REGION Network 2
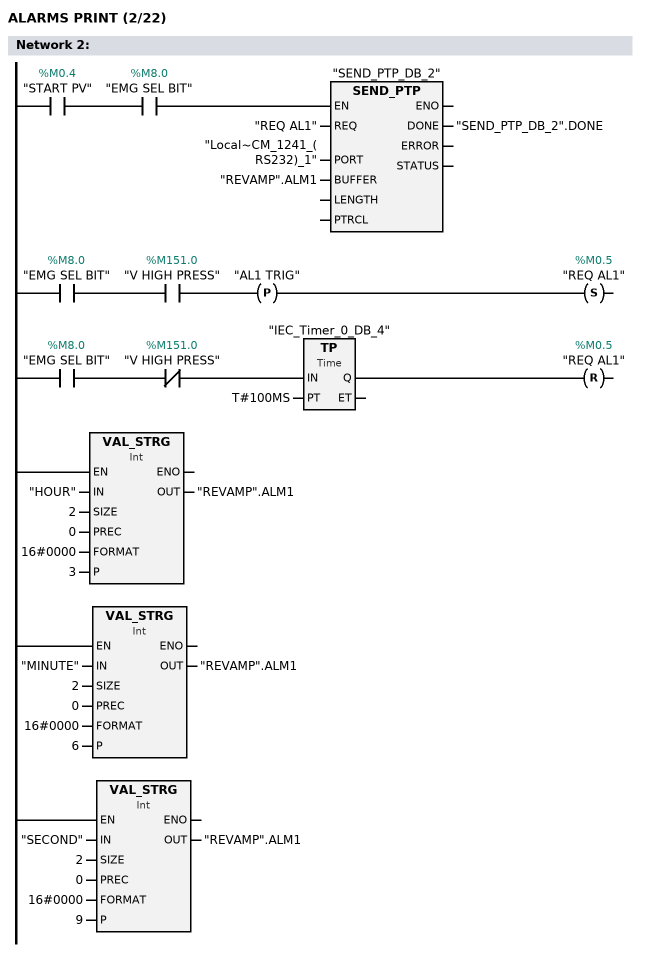
   RUNG wire#powerrail
      Contact( "START PV" )
      Contact( "EMG SEL BIT" )
      "SEND_PTP_DB_2".SEND_PTP(REQ := "REQ AL1", PORT := "Local~CM_1241_(RS232)_1", BUFFER := "REVAMP".ALM1, LENGTH :=, PTRCL :=, DONE => "SEND_PTP_DB_2".DONE, ERROR =>, STATUS =>)
   END_RUNG
   RUNG wire#powerrail
      Contact( "EMG SEL BIT" )
      Contact( "V HIGH PRESS" )
      P_Trig( "AL1 TRIG" )
      S_Coil( "REQ AL1" )
   END_RUNG
   RUNG wire#powerrail
      Contact( "EMG SEL BIT" )
      I_Contact( "V HIGH PRESS" )
      { S7_Templates := "time_type := Time" } "IEC_Timer_0_DB_4".TP(pt := T#100MS, et =>)
      R_Coil( "REQ AL1" )
   END_RUNG
   RUNG wire#powerrail
      { S7_Templates := "[value_type := Int, str_type := String]" } VAL_STRG(IN := "HOUR", SIZE := 2, PREC := 0, FORMAT := 16#0000, P := 3, OUT => "REVAMP".ALM1)
   END_RUNG
   RUNG wire#powerrail
      { S7_Templates := "[value_type := Int, str_type := String]" } VAL_STRG(IN := "MINUTE", SIZE := 2, PREC := 0, FORMAT := 16#0000, P := 6, OUT => "REVAMP".ALM1)
   END_RUNG
   RUNG wire#powerrail
      { S7_Templates := "[value_type := Int, str_type := String]" } VAL_STRG(IN := "SECOND", SIZE := 2, PREC := 0, FORMAT := 16#0000, P := 9, OUT => "REVAMP".ALM1)
   END_RUNG
   // the same network as SCL:
   IF "START PV" AND "EMG SEL BIT" THEN
       "SEND_PTP_DB_2"(REQ := "REQ AL1",   // SEND_PTP
                       PORT := "Local~CM_1241_(RS232)_1",
                       BUFFER := "REVAMP".ALM1,
                       DONE => "SEND_PTP_DB_2".DONE);
   END_IF;
   #_w1 := "EMG SEL BIT" AND "V HIGH PRESS";
   #_w2 := #_w1 AND NOT "AL1 TRIG";   // rising edge
   "AL1 TRIG" := #_w1;
   IF #_w2 THEN "REQ AL1" := TRUE; END_IF;
   "IEC_Timer_0_DB_4".TP(IN := "EMG SEL BIT" AND NOT "V HIGH PRESS", PT := T#100MS);
   IF "IEC_Timer_0_DB_4".Q THEN "REQ AL1" := FALSE; END_IF;
   VAL_STRG(IN := "HOUR", SIZE := 2, PREC := 0, FORMAT := 16#0000, P := 3, OUT => "REVAMP".ALM1);
   VAL_STRG(IN := "MINUTE", SIZE := 2, PREC := 0, FORMAT := 16#0000, P := 6, OUT => "REVAMP".ALM1);
   VAL_STRG(IN := "SECOND", SIZE := 2, PREC := 0, FORMAT := 16#0000, P := 9, OUT => "REVAMP".ALM1);
END_REGION

REGION Network 3
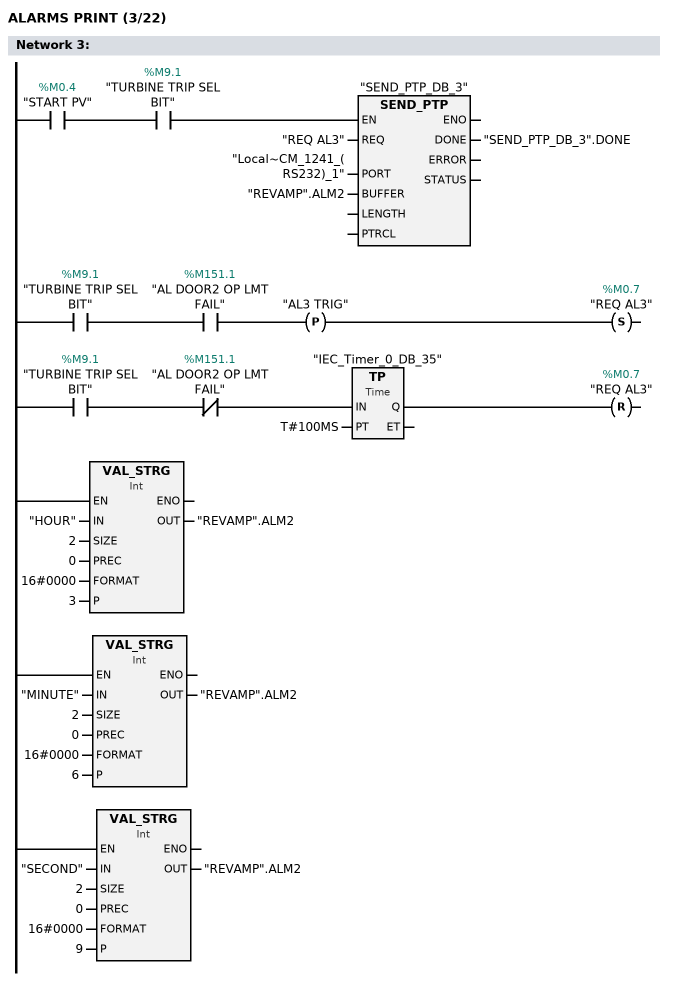
   RUNG wire#powerrail
      Contact( "START PV" )
      Contact( "TURBINE TRIP SEL BIT" )
      "SEND_PTP_DB_3".SEND_PTP(REQ := "REQ AL3", PORT := "Local~CM_1241_(RS232)_1", BUFFER := "REVAMP".ALM2, LENGTH :=, PTRCL :=, DONE => "SEND_PTP_DB_3".DONE, ERROR =>, STATUS =>)
   END_RUNG
   RUNG wire#powerrail
      Contact( "TURBINE TRIP SEL BIT" )
      Contact( "AL DOOR2 OP LMT FAIL" )
      P_Trig( "AL3 TRIG" )
      S_Coil( "REQ AL3" )
   END_RUNG
   RUNG wire#powerrail
      Contact( "TURBINE TRIP SEL BIT" )
      I_Contact( "AL DOOR2 OP LMT FAIL" )
      { S7_Templates := "time_type := Time" } "IEC_Timer_0_DB_35".TP(pt := T#100MS, et =>)
      R_Coil( "REQ AL3" )
   END_RUNG
   RUNG wire#powerrail
      { S7_Templates := "[value_type := Int, str_type := String]" } VAL_STRG(IN := "HOUR", SIZE := 2, PREC := 0, FORMAT := 16#0000, P := 3, OUT => "REVAMP".ALM2)
   END_RUNG
   RUNG wire#powerrail
      { S7_Templates := "[value_type := Int, str_type := String]" } VAL_STRG(IN := "MINUTE", SIZE := 2, PREC := 0, FORMAT := 16#0000, P := 6, OUT => "REVAMP".ALM2)
   END_RUNG
   RUNG wire#powerrail
      { S7_Templates := "[value_type := Int, str_type := String]" } VAL_STRG(IN := "SECOND", SIZE := 2, PREC := 0, FORMAT := 16#0000, P := 9, OUT => "REVAMP".ALM2)
   END_RUNG
   // the same network as SCL:
   IF "START PV" AND "TURBINE TRIP SEL BIT" THEN
       "SEND_PTP_DB_3"(REQ := "REQ AL3",   // SEND_PTP
                       PORT := "Local~CM_1241_(RS232)_1",
                       BUFFER := "REVAMP".ALM2,
                       DONE => "SEND_PTP_DB_3".DONE);
   END_IF;
   #_w1 := "TURBINE TRIP SEL BIT" AND "AL DOOR2 OP LMT FAIL";
   #_w2 := #_w1 AND NOT "AL3 TRIG";   // rising edge
   "AL3 TRIG" := #_w1;
   IF #_w2 THEN "REQ AL3" := TRUE; END_IF;
   "IEC_Timer_0_DB_35".TP(IN := "TURBINE TRIP SEL BIT" AND NOT "AL DOOR2 OP LMT FAIL", PT := T#100MS);
   IF "IEC_Timer_0_DB_35".Q THEN "REQ AL3" := FALSE; END_IF;
   VAL_STRG(IN := "HOUR", SIZE := 2, PREC := 0, FORMAT := 16#0000, P := 3, OUT => "REVAMP".ALM2);
   VAL_STRG(IN := "MINUTE", SIZE := 2, PREC := 0, FORMAT := 16#0000, P := 6, OUT => "REVAMP".ALM2);
   VAL_STRG(IN := "SECOND", SIZE := 2, PREC := 0, FORMAT := 16#0000, P := 9, OUT => "REVAMP".ALM2);
END_REGION

REGION Network 4
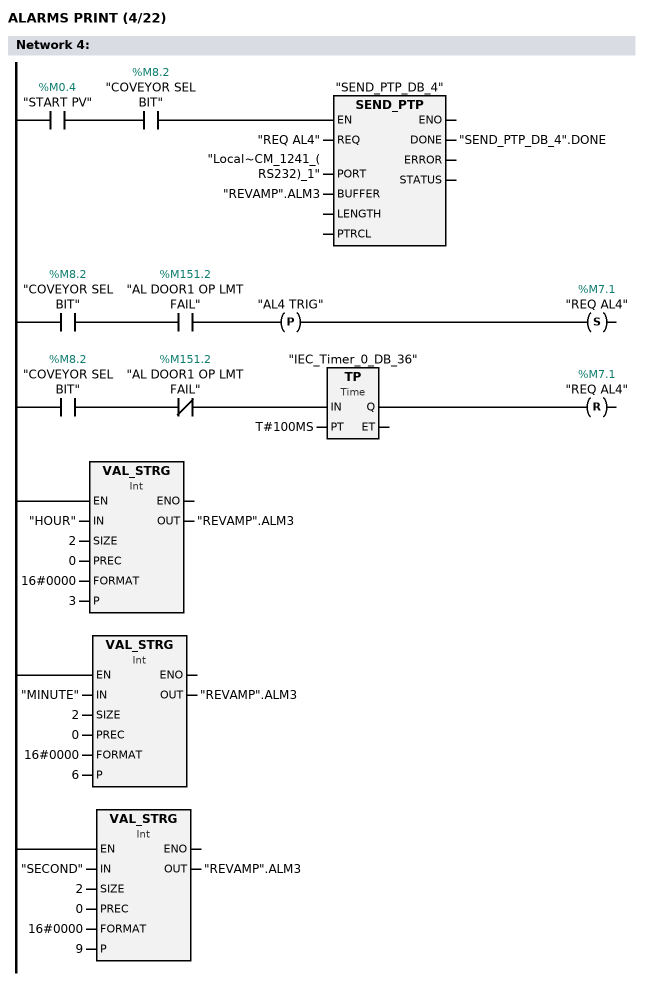
   RUNG wire#powerrail
      Contact( "START PV" )
      Contact( "COVEYOR SEL BIT" )
      "SEND_PTP_DB_4".SEND_PTP(REQ := "REQ AL4", PORT := "Local~CM_1241_(RS232)_1", BUFFER := "REVAMP".ALM3, LENGTH :=, PTRCL :=, DONE => "SEND_PTP_DB_4".DONE, ERROR =>, STATUS =>)
   END_RUNG
   RUNG wire#powerrail
      Contact( "COVEYOR SEL BIT" )
      Contact( "AL DOOR1 OP LMT FAIL" )
      P_Trig( "AL4 TRIG" )
      S_Coil( "REQ AL4" )
   END_RUNG
   RUNG wire#powerrail
      Contact( "COVEYOR SEL BIT" )
      I_Contact( "AL DOOR1 OP LMT FAIL" )
      { S7_Templates := "time_type := Time" } "IEC_Timer_0_DB_36".TP(pt := T#100MS, et =>)
      R_Coil( "REQ AL4" )
   END_RUNG
   RUNG wire#powerrail
      { S7_Templates := "[value_type := Int, str_type := String]" } VAL_STRG(IN := "HOUR", SIZE := 2, PREC := 0, FORMAT := 16#0000, P := 3, OUT => "REVAMP".ALM3)
   END_RUNG
   RUNG wire#powerrail
      { S7_Templates := "[value_type := Int, str_type := String]" } VAL_STRG(IN := "MINUTE", SIZE := 2, PREC := 0, FORMAT := 16#0000, P := 6, OUT => "REVAMP".ALM3)
   END_RUNG
   RUNG wire#powerrail
      { S7_Templates := "[value_type := Int, str_type := String]" } VAL_STRG(IN := "SECOND", SIZE := 2, PREC := 0, FORMAT := 16#0000, P := 9, OUT => "REVAMP".ALM3)
   END_RUNG
   // the same network as SCL:
   IF "START PV" AND "COVEYOR SEL BIT" THEN
       "SEND_PTP_DB_4"(REQ := "REQ AL4",   // SEND_PTP
                       PORT := "Local~CM_1241_(RS232)_1",
                       BUFFER := "REVAMP".ALM3,
                       DONE => "SEND_PTP_DB_4".DONE);
   END_IF;
   #_w1 := "COVEYOR SEL BIT" AND "AL DOOR1 OP LMT FAIL";
   #_w2 := #_w1 AND NOT "AL4 TRIG";   // rising edge
   "AL4 TRIG" := #_w1;
   IF #_w2 THEN "REQ AL4" := TRUE; END_IF;
   "IEC_Timer_0_DB_36".TP(IN := "COVEYOR SEL BIT" AND NOT "AL DOOR1 OP LMT FAIL", PT := T#100MS);
   IF "IEC_Timer_0_DB_36".Q THEN "REQ AL4" := FALSE; END_IF;
   VAL_STRG(IN := "HOUR", SIZE := 2, PREC := 0, FORMAT := 16#0000, P := 3, OUT => "REVAMP".ALM3);
   VAL_STRG(IN := "MINUTE", SIZE := 2, PREC := 0, FORMAT := 16#0000, P := 6, OUT => "REVAMP".ALM3);
   VAL_STRG(IN := "SECOND", SIZE := 2, PREC := 0, FORMAT := 16#0000, P := 9, OUT => "REVAMP".ALM3);
END_REGION

REGION Network 5
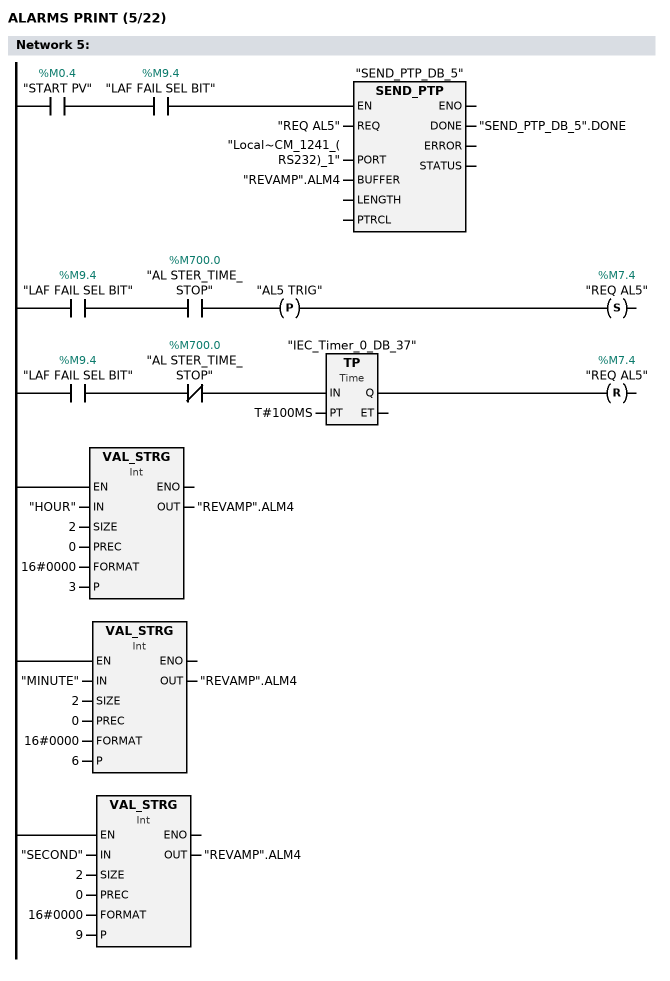
   RUNG wire#powerrail
      Contact( "START PV" )
      Contact( "LAF FAIL SEL BIT" )
      "SEND_PTP_DB_5".SEND_PTP(REQ := "REQ AL5", PORT := "Local~CM_1241_(RS232)_1", BUFFER := "REVAMP".ALM4, LENGTH :=, PTRCL :=, DONE => "SEND_PTP_DB_5".DONE, ERROR =>, STATUS =>)
   END_RUNG
   RUNG wire#powerrail
      Contact( "LAF FAIL SEL BIT" )
      Contact( "AL STER_TIME_STOP" )
      P_Trig( "AL5 TRIG" )
      S_Coil( "REQ AL5" )
   END_RUNG
   RUNG wire#powerrail
      Contact( "LAF FAIL SEL BIT" )
      I_Contact( "AL STER_TIME_STOP" )
      { S7_Templates := "time_type := Time" } "IEC_Timer_0_DB_37".TP(pt := T#100MS, et =>)
      R_Coil( "REQ AL5" )
   END_RUNG
   RUNG wire#powerrail
      { S7_Templates := "[value_type := Int, str_type := String]" } VAL_STRG(IN := "HOUR", SIZE := 2, PREC := 0, FORMAT := 16#0000, P := 3, OUT => "REVAMP".ALM4)
   END_RUNG
   RUNG wire#powerrail
      { S7_Templates := "[value_type := Int, str_type := String]" } VAL_STRG(IN := "MINUTE", SIZE := 2, PREC := 0, FORMAT := 16#0000, P := 6, OUT => "REVAMP".ALM4)
   END_RUNG
   RUNG wire#powerrail
      { S7_Templates := "[value_type := Int, str_type := String]" } VAL_STRG(IN := "SECOND", SIZE := 2, PREC := 0, FORMAT := 16#0000, P := 9, OUT => "REVAMP".ALM4)
   END_RUNG
   // the same network as SCL:
   IF "START PV" AND "LAF FAIL SEL BIT" THEN
       "SEND_PTP_DB_5"(REQ := "REQ AL5",   // SEND_PTP
                       PORT := "Local~CM_1241_(RS232)_1",
                       BUFFER := "REVAMP".ALM4,
                       DONE => "SEND_PTP_DB_5".DONE);
   END_IF;
   #_w1 := "LAF FAIL SEL BIT" AND "AL STER_TIME_STOP";
   #_w2 := #_w1 AND NOT "AL5 TRIG";   // rising edge
   "AL5 TRIG" := #_w1;
   IF #_w2 THEN "REQ AL5" := TRUE; END_IF;
   "IEC_Timer_0_DB_37".TP(IN := "LAF FAIL SEL BIT" AND NOT "AL STER_TIME_STOP", PT := T#100MS);
   IF "IEC_Timer_0_DB_37".Q THEN "REQ AL5" := FALSE; END_IF;
   VAL_STRG(IN := "HOUR", SIZE := 2, PREC := 0, FORMAT := 16#0000, P := 3, OUT => "REVAMP".ALM4);
   VAL_STRG(IN := "MINUTE", SIZE := 2, PREC := 0, FORMAT := 16#0000, P := 6, OUT => "REVAMP".ALM4);
   VAL_STRG(IN := "SECOND", SIZE := 2, PREC := 0, FORMAT := 16#0000, P := 9, OUT => "REVAMP".ALM4);
END_REGION

REGION Network 6
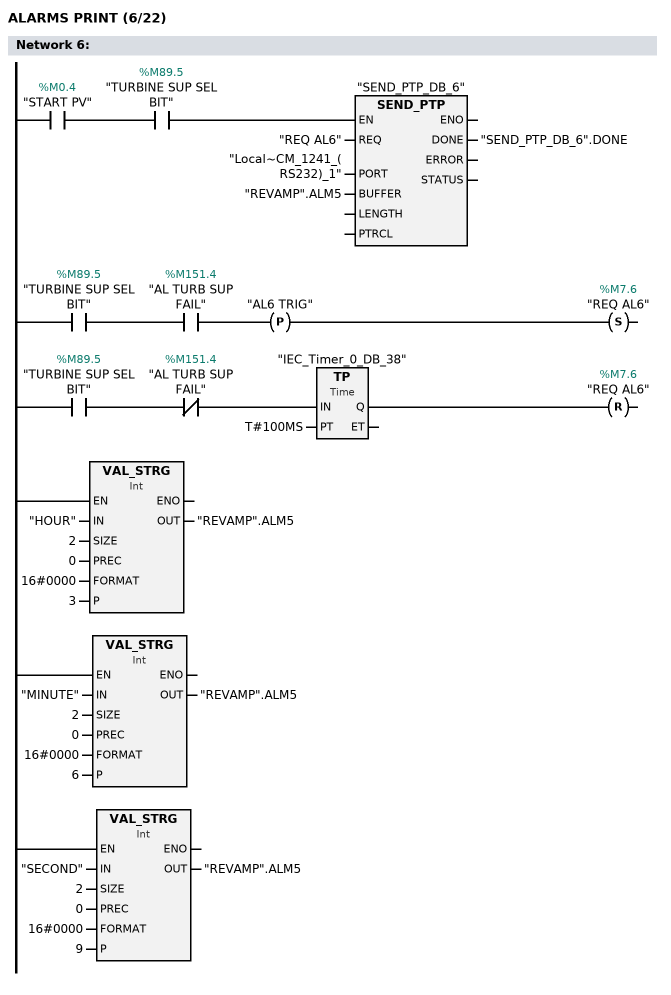
   RUNG wire#powerrail
      Contact( "START PV" )
      Contact( "TURBINE SUP SEL BIT" )
      "SEND_PTP_DB_6".SEND_PTP(REQ := "REQ AL6", PORT := "Local~CM_1241_(RS232)_1", BUFFER := "REVAMP".ALM5, LENGTH :=, PTRCL :=, DONE => "SEND_PTP_DB_6".DONE, ERROR =>, STATUS =>)
   END_RUNG
   RUNG wire#powerrail
      Contact( "TURBINE SUP SEL BIT" )
      Contact( "AL TURB SUP FAIL" )
      P_Trig( "AL6 TRIG" )
      S_Coil( "REQ AL6" )
   END_RUNG
   RUNG wire#powerrail
      Contact( "TURBINE SUP SEL BIT" )
      I_Contact( "AL TURB SUP FAIL" )
      { S7_Templates := "time_type := Time" } "IEC_Timer_0_DB_38".TP(pt := T#100MS, et =>)
      R_Coil( "REQ AL6" )
   END_RUNG
   RUNG wire#powerrail
      { S7_Templates := "[value_type := Int, str_type := String]" } VAL_STRG(IN := "HOUR", SIZE := 2, PREC := 0, FORMAT := 16#0000, P := 3, OUT => "REVAMP".ALM5)
   END_RUNG
   RUNG wire#powerrail
      { S7_Templates := "[value_type := Int, str_type := String]" } VAL_STRG(IN := "MINUTE", SIZE := 2, PREC := 0, FORMAT := 16#0000, P := 6, OUT => "REVAMP".ALM5)
   END_RUNG
   RUNG wire#powerrail
      { S7_Templates := "[value_type := Int, str_type := String]" } VAL_STRG(IN := "SECOND", SIZE := 2, PREC := 0, FORMAT := 16#0000, P := 9, OUT => "REVAMP".ALM5)
   END_RUNG
   // the same network as SCL:
   IF "START PV" AND "TURBINE SUP SEL BIT" THEN
       "SEND_PTP_DB_6"(REQ := "REQ AL6",   // SEND_PTP
                       PORT := "Local~CM_1241_(RS232)_1",
                       BUFFER := "REVAMP".ALM5,
                       DONE => "SEND_PTP_DB_6".DONE);
   END_IF;
   #_w1 := "TURBINE SUP SEL BIT" AND "AL TURB SUP FAIL";
   #_w2 := #_w1 AND NOT "AL6 TRIG";   // rising edge
   "AL6 TRIG" := #_w1;
   IF #_w2 THEN "REQ AL6" := TRUE; END_IF;
   "IEC_Timer_0_DB_38".TP(IN := "TURBINE SUP SEL BIT" AND NOT "AL TURB SUP FAIL", PT := T#100MS);
   IF "IEC_Timer_0_DB_38".Q THEN "REQ AL6" := FALSE; END_IF;
   VAL_STRG(IN := "HOUR", SIZE := 2, PREC := 0, FORMAT := 16#0000, P := 3, OUT => "REVAMP".ALM5);
   VAL_STRG(IN := "MINUTE", SIZE := 2, PREC := 0, FORMAT := 16#0000, P := 6, OUT => "REVAMP".ALM5);
   VAL_STRG(IN := "SECOND", SIZE := 2, PREC := 0, FORMAT := 16#0000, P := 9, OUT => "REVAMP".ALM5);
END_REGION

REGION Network 7
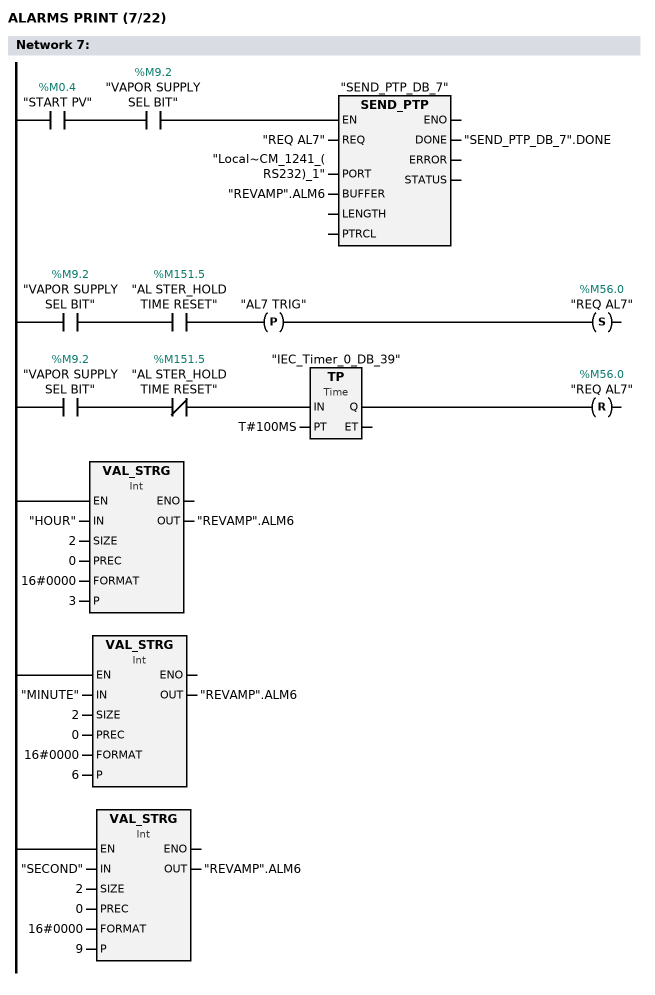
   RUNG wire#powerrail
      Contact( "START PV" )
      Contact( "VAPOR SUPPLY SEL BIT" )
      "SEND_PTP_DB_7".SEND_PTP(REQ := "REQ AL7", PORT := "Local~CM_1241_(RS232)_1", BUFFER := "REVAMP".ALM6, LENGTH :=, PTRCL :=, DONE => "SEND_PTP_DB_7".DONE, ERROR =>, STATUS =>)
   END_RUNG
   RUNG wire#powerrail
      Contact( "VAPOR SUPPLY SEL BIT" )
      Contact( "AL STER_HOLD TIME RESET" )
      P_Trig( "AL7 TRIG" )
      S_Coil( "REQ AL7" )
   END_RUNG
   RUNG wire#powerrail
      Contact( "VAPOR SUPPLY SEL BIT" )
      I_Contact( "AL STER_HOLD TIME RESET" )
      { S7_Templates := "time_type := Time" } "IEC_Timer_0_DB_39".TP(pt := T#100MS, et =>)
      R_Coil( "REQ AL7" )
   END_RUNG
   RUNG wire#powerrail
      { S7_Templates := "[value_type := Int, str_type := String]" } VAL_STRG(IN := "HOUR", SIZE := 2, PREC := 0, FORMAT := 16#0000, P := 3, OUT => "REVAMP".ALM6)
   END_RUNG
   RUNG wire#powerrail
      { S7_Templates := "[value_type := Int, str_type := String]" } VAL_STRG(IN := "MINUTE", SIZE := 2, PREC := 0, FORMAT := 16#0000, P := 6, OUT => "REVAMP".ALM6)
   END_RUNG
   RUNG wire#powerrail
      { S7_Templates := "[value_type := Int, str_type := String]" } VAL_STRG(IN := "SECOND", SIZE := 2, PREC := 0, FORMAT := 16#0000, P := 9, OUT => "REVAMP".ALM6)
   END_RUNG
   // the same network as SCL:
   IF "START PV" AND "VAPOR SUPPLY SEL BIT" THEN
       "SEND_PTP_DB_7"(REQ := "REQ AL7",   // SEND_PTP
                       PORT := "Local~CM_1241_(RS232)_1",
                       BUFFER := "REVAMP".ALM6,
                       DONE => "SEND_PTP_DB_7".DONE);
   END_IF;
   #_w1 := "VAPOR SUPPLY SEL BIT" AND "AL STER_HOLD TIME RESET";
   #_w2 := #_w1 AND NOT "AL7 TRIG";   // rising edge
   "AL7 TRIG" := #_w1;
   IF #_w2 THEN "REQ AL7" := TRUE; END_IF;
   "IEC_Timer_0_DB_39".TP(IN := "VAPOR SUPPLY SEL BIT" AND NOT "AL STER_HOLD TIME RESET", PT := T#100MS);
   IF "IEC_Timer_0_DB_39".Q THEN "REQ AL7" := FALSE; END_IF;
   VAL_STRG(IN := "HOUR", SIZE := 2, PREC := 0, FORMAT := 16#0000, P := 3, OUT => "REVAMP".ALM6);
   VAL_STRG(IN := "MINUTE", SIZE := 2, PREC := 0, FORMAT := 16#0000, P := 6, OUT => "REVAMP".ALM6);
   VAL_STRG(IN := "SECOND", SIZE := 2, PREC := 0, FORMAT := 16#0000, P := 9, OUT => "REVAMP".ALM6);
END_REGION

REGION Network 8
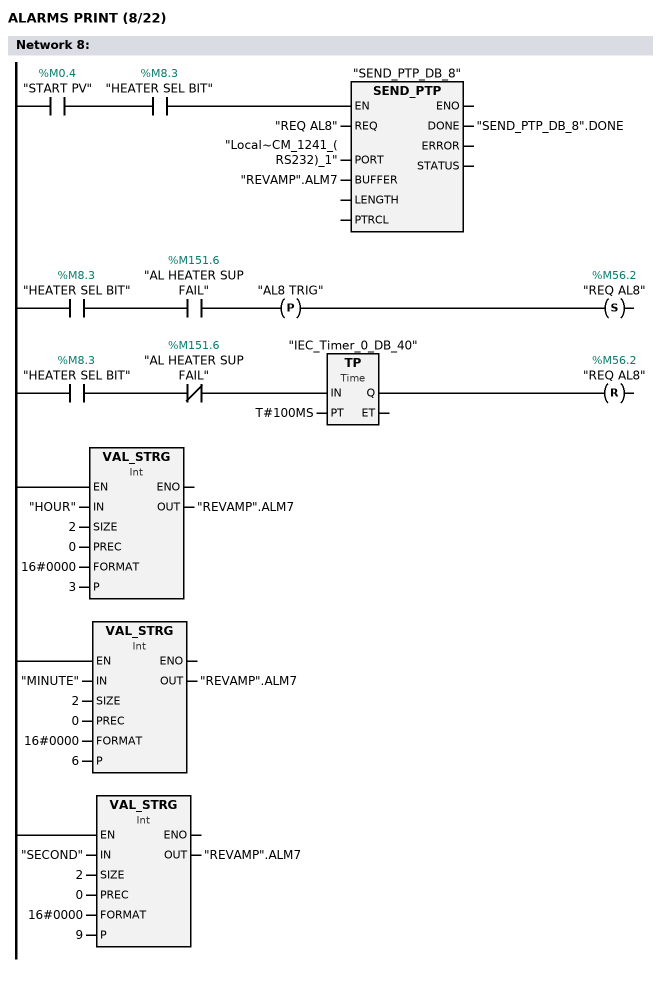
   RUNG wire#powerrail
      Contact( "START PV" )
      Contact( "HEATER SEL BIT" )
      "SEND_PTP_DB_8".SEND_PTP(REQ := "REQ AL8", PORT := "Local~CM_1241_(RS232)_1", BUFFER := "REVAMP".ALM7, LENGTH :=, PTRCL :=, DONE => "SEND_PTP_DB_8".DONE, ERROR =>, STATUS =>)
   END_RUNG
   RUNG wire#powerrail
      Contact( "HEATER SEL BIT" )
      Contact( "AL HEATER SUP FAIL" )
      P_Trig( "AL8 TRIG" )
      S_Coil( "REQ AL8" )
   END_RUNG
   RUNG wire#powerrail
      Contact( "HEATER SEL BIT" )
      I_Contact( "AL HEATER SUP FAIL" )
      { S7_Templates := "time_type := Time" } "IEC_Timer_0_DB_40".TP(pt := T#100MS, et =>)
      R_Coil( "REQ AL8" )
   END_RUNG
   RUNG wire#powerrail
      { S7_Templates := "[value_type := Int, str_type := String]" } VAL_STRG(IN := "HOUR", SIZE := 2, PREC := 0, FORMAT := 16#0000, P := 3, OUT => "REVAMP".ALM7)
   END_RUNG
   RUNG wire#powerrail
      { S7_Templates := "[value_type := Int, str_type := String]" } VAL_STRG(IN := "MINUTE", SIZE := 2, PREC := 0, FORMAT := 16#0000, P := 6, OUT => "REVAMP".ALM7)
   END_RUNG
   RUNG wire#powerrail
      { S7_Templates := "[value_type := Int, str_type := String]" } VAL_STRG(IN := "SECOND", SIZE := 2, PREC := 0, FORMAT := 16#0000, P := 9, OUT => "REVAMP".ALM7)
   END_RUNG
   // the same network as SCL:
   IF "START PV" AND "HEATER SEL BIT" THEN
       "SEND_PTP_DB_8"(REQ := "REQ AL8",   // SEND_PTP
                       PORT := "Local~CM_1241_(RS232)_1",
                       BUFFER := "REVAMP".ALM7,
                       DONE => "SEND_PTP_DB_8".DONE);
   END_IF;
   #_w1 := "HEATER SEL BIT" AND "AL HEATER SUP FAIL";
   #_w2 := #_w1 AND NOT "AL8 TRIG";   // rising edge
   "AL8 TRIG" := #_w1;
   IF #_w2 THEN "REQ AL8" := TRUE; END_IF;
   "IEC_Timer_0_DB_40".TP(IN := "HEATER SEL BIT" AND NOT "AL HEATER SUP FAIL", PT := T#100MS);
   IF "IEC_Timer_0_DB_40".Q THEN "REQ AL8" := FALSE; END_IF;
   VAL_STRG(IN := "HOUR", SIZE := 2, PREC := 0, FORMAT := 16#0000, P := 3, OUT => "REVAMP".ALM7);
   VAL_STRG(IN := "MINUTE", SIZE := 2, PREC := 0, FORMAT := 16#0000, P := 6, OUT => "REVAMP".ALM7);
   VAL_STRG(IN := "SECOND", SIZE := 2, PREC := 0, FORMAT := 16#0000, P := 9, OUT => "REVAMP".ALM7);
END_REGION

REGION Network 9
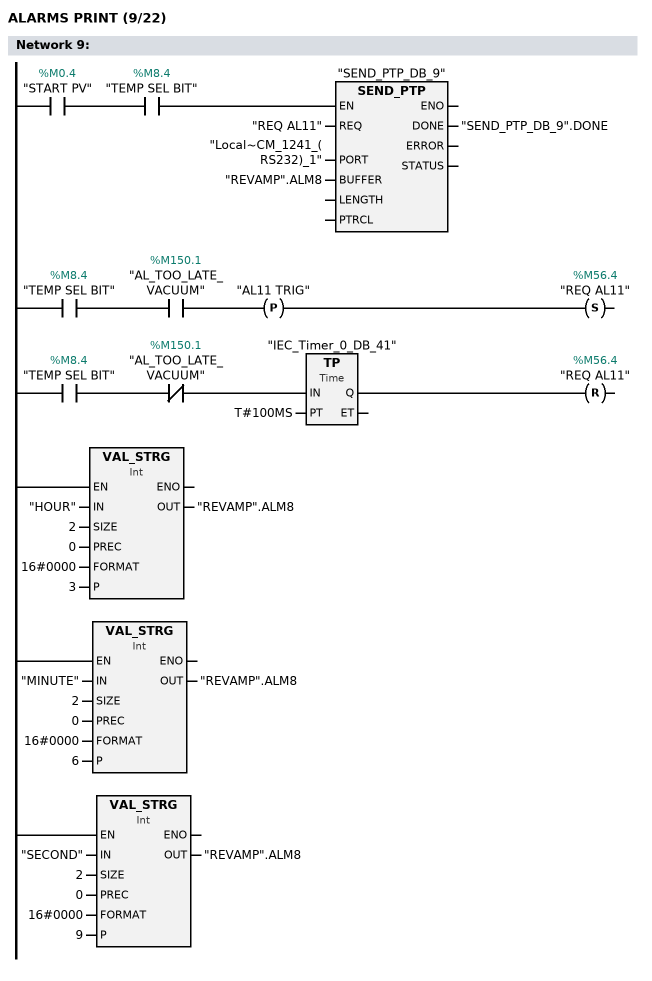
   RUNG wire#powerrail
      Contact( "START PV" )
      Contact( "TEMP SEL BIT" )
      "SEND_PTP_DB_9".SEND_PTP(REQ := "REQ AL11", PORT := "Local~CM_1241_(RS232)_1", BUFFER := "REVAMP".ALM8, LENGTH :=, PTRCL :=, DONE => "SEND_PTP_DB_9".DONE, ERROR =>, STATUS =>)
   END_RUNG
   RUNG wire#powerrail
      Contact( "TEMP SEL BIT" )
      Contact( "AL_TOO_LATE_VACUUM" )
      P_Trig( "AL11 TRIG" )
      S_Coil( "REQ AL11" )
   END_RUNG
   RUNG wire#powerrail
      Contact( "TEMP SEL BIT" )
      I_Contact( "AL_TOO_LATE_VACUUM" )
      { S7_Templates := "time_type := Time" } "IEC_Timer_0_DB_41".TP(pt := T#100MS, et =>)
      R_Coil( "REQ AL11" )
   END_RUNG
   RUNG wire#powerrail
      { S7_Templates := "[value_type := Int, str_type := String]" } VAL_STRG(IN := "HOUR", SIZE := 2, PREC := 0, FORMAT := 16#0000, P := 3, OUT => "REVAMP".ALM8)
   END_RUNG
   RUNG wire#powerrail
      { S7_Templates := "[value_type := Int, str_type := String]" } VAL_STRG(IN := "MINUTE", SIZE := 2, PREC := 0, FORMAT := 16#0000, P := 6, OUT => "REVAMP".ALM8)
   END_RUNG
   RUNG wire#powerrail
      { S7_Templates := "[value_type := Int, str_type := String]" } VAL_STRG(IN := "SECOND", SIZE := 2, PREC := 0, FORMAT := 16#0000, P := 9, OUT => "REVAMP".ALM8)
   END_RUNG
   // the same network as SCL:
   IF "START PV" AND "TEMP SEL BIT" THEN
       "SEND_PTP_DB_9"(REQ := "REQ AL11",   // SEND_PTP
                       PORT := "Local~CM_1241_(RS232)_1",
                       BUFFER := "REVAMP".ALM8,
                       DONE => "SEND_PTP_DB_9".DONE);
   END_IF;
   #_w1 := "TEMP SEL BIT" AND "AL_TOO_LATE_VACUUM";
   #_w2 := #_w1 AND NOT "AL11 TRIG";   // rising edge
   "AL11 TRIG" := #_w1;
   IF #_w2 THEN "REQ AL11" := TRUE; END_IF;
   "IEC_Timer_0_DB_41".TP(IN := "TEMP SEL BIT" AND NOT "AL_TOO_LATE_VACUUM", PT := T#100MS);
   IF "IEC_Timer_0_DB_41".Q THEN "REQ AL11" := FALSE; END_IF;
   VAL_STRG(IN := "HOUR", SIZE := 2, PREC := 0, FORMAT := 16#0000, P := 3, OUT => "REVAMP".ALM8);
   VAL_STRG(IN := "MINUTE", SIZE := 2, PREC := 0, FORMAT := 16#0000, P := 6, OUT => "REVAMP".ALM8);
   VAL_STRG(IN := "SECOND", SIZE := 2, PREC := 0, FORMAT := 16#0000, P := 9, OUT => "REVAMP".ALM8);
END_REGION

REGION Network 10
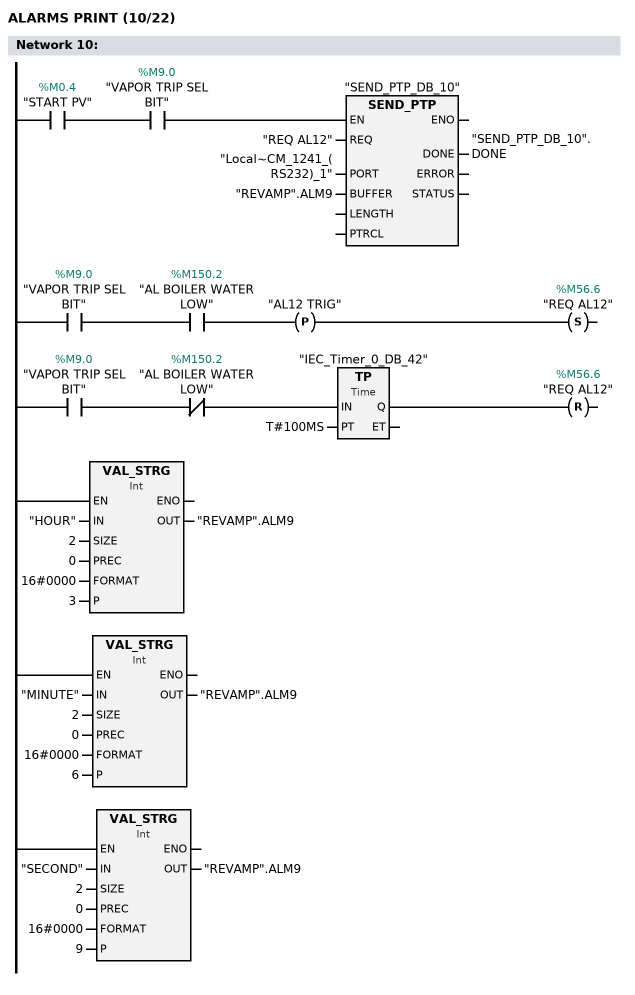
   RUNG wire#powerrail
      Contact( "START PV" )
      Contact( "VAPOR TRIP SEL BIT" )
      "SEND_PTP_DB_10".SEND_PTP(REQ := "REQ AL12", PORT := "Local~CM_1241_(RS232)_1", BUFFER := "REVAMP".ALM9, LENGTH :=, PTRCL :=, DONE => "SEND_PTP_DB_10".DONE, ERROR =>, STATUS =>)
   END_RUNG
   RUNG wire#powerrail
      Contact( "VAPOR TRIP SEL BIT" )
      Contact( "AL BOILER WATER LOW" )
      P_Trig( "AL12 TRIG" )
      S_Coil( "REQ AL12" )
   END_RUNG
   RUNG wire#powerrail
      Contact( "VAPOR TRIP SEL BIT" )
      I_Contact( "AL BOILER WATER LOW" )
      { S7_Templates := "time_type := Time" } "IEC_Timer_0_DB_42".TP(pt := T#100MS, et =>)
      R_Coil( "REQ AL12" )
   END_RUNG
   RUNG wire#powerrail
      { S7_Templates := "[value_type := Int, str_type := String]" } VAL_STRG(IN := "HOUR", SIZE := 2, PREC := 0, FORMAT := 16#0000, P := 3, OUT => "REVAMP".ALM9)
   END_RUNG
   RUNG wire#powerrail
      { S7_Templates := "[value_type := Int, str_type := String]" } VAL_STRG(IN := "MINUTE", SIZE := 2, PREC := 0, FORMAT := 16#0000, P := 6, OUT => "REVAMP".ALM9)
   END_RUNG
   RUNG wire#powerrail
      { S7_Templates := "[value_type := Int, str_type := String]" } VAL_STRG(IN := "SECOND", SIZE := 2, PREC := 0, FORMAT := 16#0000, P := 9, OUT => "REVAMP".ALM9)
   END_RUNG
   // the same network as SCL:
   IF "START PV" AND "VAPOR TRIP SEL BIT" THEN
       "SEND_PTP_DB_10"(REQ := "REQ AL12",   // SEND_PTP
                        PORT := "Local~CM_1241_(RS232)_1",
                        BUFFER := "REVAMP".ALM9,
                        DONE => "SEND_PTP_DB_10".DONE);
   END_IF;
   #_w1 := "VAPOR TRIP SEL BIT" AND "AL BOILER WATER LOW";
   #_w2 := #_w1 AND NOT "AL12 TRIG";   // rising edge
   "AL12 TRIG" := #_w1;
   IF #_w2 THEN "REQ AL12" := TRUE; END_IF;
   "IEC_Timer_0_DB_42".TP(IN := "VAPOR TRIP SEL BIT" AND NOT "AL BOILER WATER LOW", PT := T#100MS);
   IF "IEC_Timer_0_DB_42".Q THEN "REQ AL12" := FALSE; END_IF;
   VAL_STRG(IN := "HOUR", SIZE := 2, PREC := 0, FORMAT := 16#0000, P := 3, OUT => "REVAMP".ALM9);
   VAL_STRG(IN := "MINUTE", SIZE := 2, PREC := 0, FORMAT := 16#0000, P := 6, OUT => "REVAMP".ALM9);
   VAL_STRG(IN := "SECOND", SIZE := 2, PREC := 0, FORMAT := 16#0000, P := 9, OUT => "REVAMP".ALM9);
END_REGION

REGION Network 11
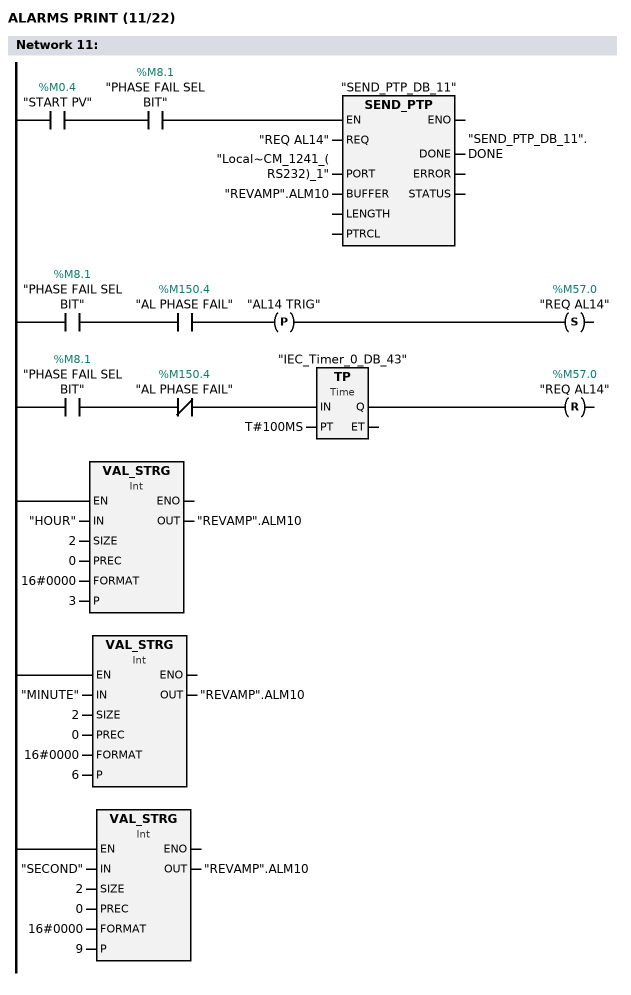
   RUNG wire#powerrail
      Contact( "START PV" )
      Contact( "PHASE FAIL SEL BIT" )
      "SEND_PTP_DB_11".SEND_PTP(REQ := "REQ AL14", PORT := "Local~CM_1241_(RS232)_1", BUFFER := "REVAMP".ALM10, LENGTH :=, PTRCL :=, DONE => "SEND_PTP_DB_11".DONE, ERROR =>, STATUS =>)
   END_RUNG
   RUNG wire#powerrail
      Contact( "PHASE FAIL SEL BIT" )
      Contact( "AL PHASE FAIL" )
      P_Trig( "AL14 TRIG" )
      S_Coil( "REQ AL14" )
   END_RUNG
   RUNG wire#powerrail
      Contact( "PHASE FAIL SEL BIT" )
      I_Contact( "AL PHASE FAIL" )
      { S7_Templates := "time_type := Time" } "IEC_Timer_0_DB_43".TP(pt := T#100MS, et =>)
      R_Coil( "REQ AL14" )
   END_RUNG
   RUNG wire#powerrail
      { S7_Templates := "[value_type := Int, str_type := String]" } VAL_STRG(IN := "HOUR", SIZE := 2, PREC := 0, FORMAT := 16#0000, P := 3, OUT => "REVAMP".ALM10)
   END_RUNG
   RUNG wire#powerrail
      { S7_Templates := "[value_type := Int, str_type := String]" } VAL_STRG(IN := "MINUTE", SIZE := 2, PREC := 0, FORMAT := 16#0000, P := 6, OUT => "REVAMP".ALM10)
   END_RUNG
   RUNG wire#powerrail
      { S7_Templates := "[value_type := Int, str_type := String]" } VAL_STRG(IN := "SECOND", SIZE := 2, PREC := 0, FORMAT := 16#0000, P := 9, OUT => "REVAMP".ALM10)
   END_RUNG
   // the same network as SCL:
   IF "START PV" AND "PHASE FAIL SEL BIT" THEN
       "SEND_PTP_DB_11"(REQ := "REQ AL14",   // SEND_PTP
                        PORT := "Local~CM_1241_(RS232)_1",
                        BUFFER := "REVAMP".ALM10,
                        DONE => "SEND_PTP_DB_11".DONE);
   END_IF;
   #_w1 := "PHASE FAIL SEL BIT" AND "AL PHASE FAIL";
   #_w2 := #_w1 AND NOT "AL14 TRIG";   // rising edge
   "AL14 TRIG" := #_w1;
   IF #_w2 THEN "REQ AL14" := TRUE; END_IF;
   "IEC_Timer_0_DB_43".TP(IN := "PHASE FAIL SEL BIT" AND NOT "AL PHASE FAIL", PT := T#100MS);
   IF "IEC_Timer_0_DB_43".Q THEN "REQ AL14" := FALSE; END_IF;
   VAL_STRG(IN := "HOUR", SIZE := 2, PREC := 0, FORMAT := 16#0000, P := 3, OUT => "REVAMP".ALM10);
   VAL_STRG(IN := "MINUTE", SIZE := 2, PREC := 0, FORMAT := 16#0000, P := 6, OUT => "REVAMP".ALM10);
   VAL_STRG(IN := "SECOND", SIZE := 2, PREC := 0, FORMAT := 16#0000, P := 9, OUT => "REVAMP".ALM10);
END_REGION

REGION Network 12
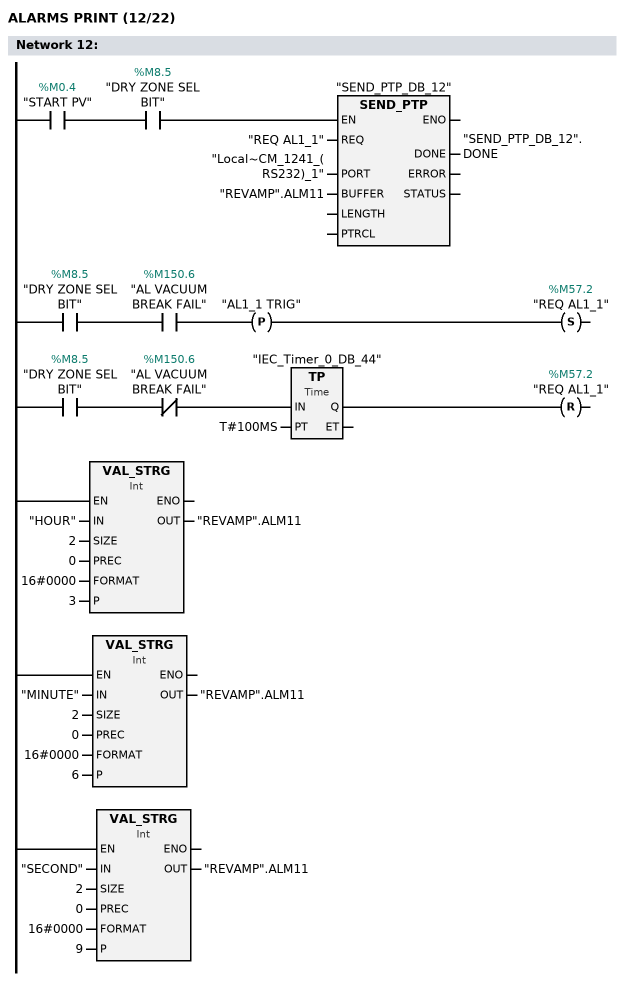
   RUNG wire#powerrail
      Contact( "START PV" )
      Contact( "DRY ZONE SEL BIT" )
      "SEND_PTP_DB_12".SEND_PTP(REQ := "REQ AL1_1", PORT := "Local~CM_1241_(RS232)_1", BUFFER := "REVAMP".ALM11, LENGTH :=, PTRCL :=, DONE => "SEND_PTP_DB_12".DONE, ERROR =>, STATUS =>)
   END_RUNG
   RUNG wire#powerrail
      Contact( "DRY ZONE SEL BIT" )
      Contact( "AL VACUUM BREAK FAIL" )
      P_Trig( "AL1_1 TRIG" )
      S_Coil( "REQ AL1_1" )
   END_RUNG
   RUNG wire#powerrail
      Contact( "DRY ZONE SEL BIT" )
      I_Contact( "AL VACUUM BREAK FAIL" )
      { S7_Templates := "time_type := Time" } "IEC_Timer_0_DB_44".TP(pt := T#100MS, et =>)
      R_Coil( "REQ AL1_1" )
   END_RUNG
   RUNG wire#powerrail
      { S7_Templates := "[value_type := Int, str_type := String]" } VAL_STRG(IN := "HOUR", SIZE := 2, PREC := 0, FORMAT := 16#0000, P := 3, OUT => "REVAMP".ALM11)
   END_RUNG
   RUNG wire#powerrail
      { S7_Templates := "[value_type := Int, str_type := String]" } VAL_STRG(IN := "MINUTE", SIZE := 2, PREC := 0, FORMAT := 16#0000, P := 6, OUT => "REVAMP".ALM11)
   END_RUNG
   RUNG wire#powerrail
      { S7_Templates := "[value_type := Int, str_type := String]" } VAL_STRG(IN := "SECOND", SIZE := 2, PREC := 0, FORMAT := 16#0000, P := 9, OUT => "REVAMP".ALM11)
   END_RUNG
   // the same network as SCL:
   IF "START PV" AND "DRY ZONE SEL BIT" THEN
       "SEND_PTP_DB_12"(REQ := "REQ AL1_1",   // SEND_PTP
                        PORT := "Local~CM_1241_(RS232)_1",
                        BUFFER := "REVAMP".ALM11,
                        DONE => "SEND_PTP_DB_12".DONE);
   END_IF;
   #_w1 := "DRY ZONE SEL BIT" AND "AL VACUUM BREAK FAIL";
   #_w2 := #_w1 AND NOT "AL1_1 TRIG";   // rising edge
   "AL1_1 TRIG" := #_w1;
   IF #_w2 THEN "REQ AL1_1" := TRUE; END_IF;
   "IEC_Timer_0_DB_44".TP(IN := "DRY ZONE SEL BIT" AND NOT "AL VACUUM BREAK FAIL", PT := T#100MS);
   IF "IEC_Timer_0_DB_44".Q THEN "REQ AL1_1" := FALSE; END_IF;
   VAL_STRG(IN := "HOUR", SIZE := 2, PREC := 0, FORMAT := 16#0000, P := 3, OUT => "REVAMP".ALM11);
   VAL_STRG(IN := "MINUTE", SIZE := 2, PREC := 0, FORMAT := 16#0000, P := 6, OUT => "REVAMP".ALM11);
   VAL_STRG(IN := "SECOND", SIZE := 2, PREC := 0, FORMAT := 16#0000, P := 9, OUT => "REVAMP".ALM11);
END_REGION

REGION Network 13
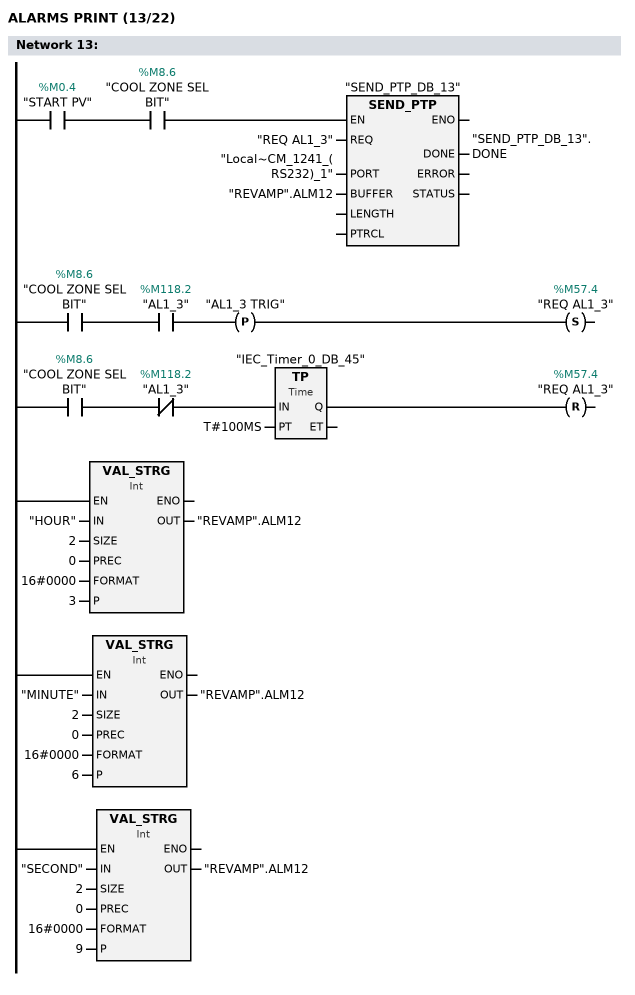
   RUNG wire#powerrail
      Contact( "START PV" )
      Contact( "COOL ZONE SEL BIT" )
      "SEND_PTP_DB_13".SEND_PTP(REQ := "REQ AL1_3", PORT := "Local~CM_1241_(RS232)_1", BUFFER := "REVAMP".ALM12, LENGTH :=, PTRCL :=, DONE => "SEND_PTP_DB_13".DONE, ERROR =>, STATUS =>)
   END_RUNG
   RUNG wire#powerrail
      Contact( "COOL ZONE SEL BIT" )
      Contact( "AL1_3" )
      P_Trig( "AL1_3 TRIG" )
      S_Coil( "REQ AL1_3" )
   END_RUNG
   RUNG wire#powerrail
      Contact( "COOL ZONE SEL BIT" )
      I_Contact( "AL1_3" )
      { S7_Templates := "time_type := Time" } "IEC_Timer_0_DB_45".TP(pt := T#100MS, et =>)
      R_Coil( "REQ AL1_3" )
   END_RUNG
   RUNG wire#powerrail
      { S7_Templates := "[value_type := Int, str_type := String]" } VAL_STRG(IN := "HOUR", SIZE := 2, PREC := 0, FORMAT := 16#0000, P := 3, OUT => "REVAMP".ALM12)
   END_RUNG
   RUNG wire#powerrail
      { S7_Templates := "[value_type := Int, str_type := String]" } VAL_STRG(IN := "MINUTE", SIZE := 2, PREC := 0, FORMAT := 16#0000, P := 6, OUT => "REVAMP".ALM12)
   END_RUNG
   RUNG wire#powerrail
      { S7_Templates := "[value_type := Int, str_type := String]" } VAL_STRG(IN := "SECOND", SIZE := 2, PREC := 0, FORMAT := 16#0000, P := 9, OUT => "REVAMP".ALM12)
   END_RUNG
   // the same network as SCL:
   IF "START PV" AND "COOL ZONE SEL BIT" THEN
       "SEND_PTP_DB_13"(REQ := "REQ AL1_3",   // SEND_PTP
                        PORT := "Local~CM_1241_(RS232)_1",
                        BUFFER := "REVAMP".ALM12,
                        DONE => "SEND_PTP_DB_13".DONE);
   END_IF;
   #_w1 := "COOL ZONE SEL BIT" AND "AL1_3";
   #_w2 := #_w1 AND NOT "AL1_3 TRIG";   // rising edge
   "AL1_3 TRIG" := #_w1;
   IF #_w2 THEN "REQ AL1_3" := TRUE; END_IF;
   "IEC_Timer_0_DB_45".TP(IN := "COOL ZONE SEL BIT" AND NOT "AL1_3", PT := T#100MS);
   IF "IEC_Timer_0_DB_45".Q THEN "REQ AL1_3" := FALSE; END_IF;
   VAL_STRG(IN := "HOUR", SIZE := 2, PREC := 0, FORMAT := 16#0000, P := 3, OUT => "REVAMP".ALM12);
   VAL_STRG(IN := "MINUTE", SIZE := 2, PREC := 0, FORMAT := 16#0000, P := 6, OUT => "REVAMP".ALM12);
   VAL_STRG(IN := "SECOND", SIZE := 2, PREC := 0, FORMAT := 16#0000, P := 9, OUT => "REVAMP".ALM12);
END_REGION

REGION Network 14
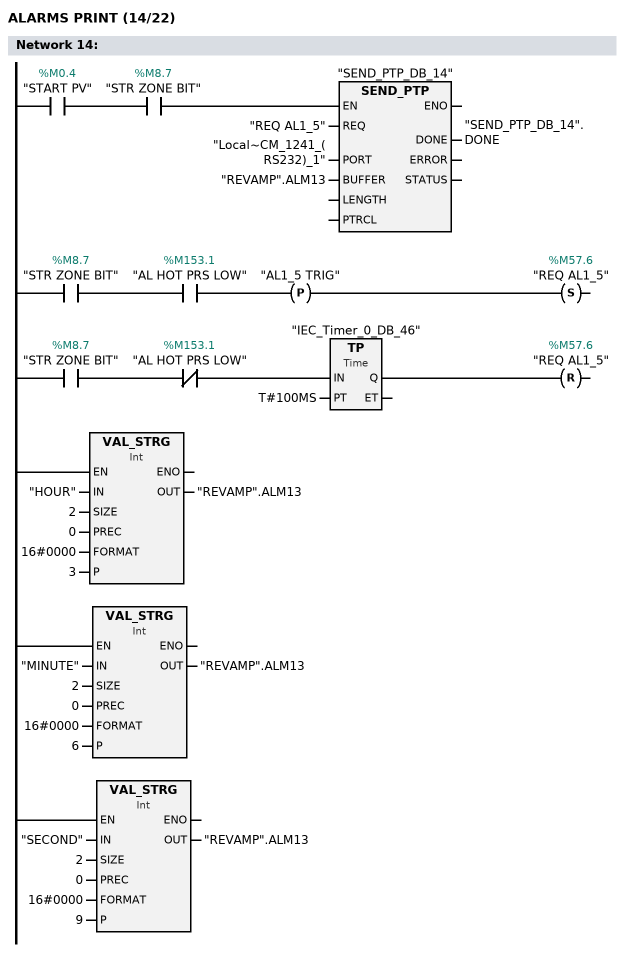
   RUNG wire#powerrail
      Contact( "START PV" )
      Contact( "STR ZONE BIT" )
      "SEND_PTP_DB_14".SEND_PTP(REQ := "REQ AL1_5", PORT := "Local~CM_1241_(RS232)_1", BUFFER := "REVAMP".ALM13, LENGTH :=, PTRCL :=, DONE => "SEND_PTP_DB_14".DONE, ERROR =>, STATUS =>)
   END_RUNG
   RUNG wire#powerrail
      Contact( "STR ZONE BIT" )
      Contact( "AL HOT PRS LOW" )
      P_Trig( "AL1_5 TRIG" )
      S_Coil( "REQ AL1_5" )
   END_RUNG
   RUNG wire#powerrail
      Contact( "STR ZONE BIT" )
      I_Contact( "AL HOT PRS LOW" )
      { S7_Templates := "time_type := Time" } "IEC_Timer_0_DB_46".TP(pt := T#100MS, et =>)
      R_Coil( "REQ AL1_5" )
   END_RUNG
   RUNG wire#powerrail
      { S7_Templates := "[value_type := Int, str_type := String]" } VAL_STRG(IN := "HOUR", SIZE := 2, PREC := 0, FORMAT := 16#0000, P := 3, OUT => "REVAMP".ALM13)
   END_RUNG
   RUNG wire#powerrail
      { S7_Templates := "[value_type := Int, str_type := String]" } VAL_STRG(IN := "MINUTE", SIZE := 2, PREC := 0, FORMAT := 16#0000, P := 6, OUT => "REVAMP".ALM13)
   END_RUNG
   RUNG wire#powerrail
      { S7_Templates := "[value_type := Int, str_type := String]" } VAL_STRG(IN := "SECOND", SIZE := 2, PREC := 0, FORMAT := 16#0000, P := 9, OUT => "REVAMP".ALM13)
   END_RUNG
   // the same network as SCL:
   IF "START PV" AND "STR ZONE BIT" THEN
       "SEND_PTP_DB_14"(REQ := "REQ AL1_5",   // SEND_PTP
                        PORT := "Local~CM_1241_(RS232)_1",
                        BUFFER := "REVAMP".ALM13,
                        DONE => "SEND_PTP_DB_14".DONE);
   END_IF;
   #_w1 := "STR ZONE BIT" AND "AL HOT PRS LOW";
   #_w2 := #_w1 AND NOT "AL1_5 TRIG";   // rising edge
   "AL1_5 TRIG" := #_w1;
   IF #_w2 THEN "REQ AL1_5" := TRUE; END_IF;
   "IEC_Timer_0_DB_46".TP(IN := "STR ZONE BIT" AND NOT "AL HOT PRS LOW", PT := T#100MS);
   IF "IEC_Timer_0_DB_46".Q THEN "REQ AL1_5" := FALSE; END_IF;
   VAL_STRG(IN := "HOUR", SIZE := 2, PREC := 0, FORMAT := 16#0000, P := 3, OUT => "REVAMP".ALM13);
   VAL_STRG(IN := "MINUTE", SIZE := 2, PREC := 0, FORMAT := 16#0000, P := 6, OUT => "REVAMP".ALM13);
   VAL_STRG(IN := "SECOND", SIZE := 2, PREC := 0, FORMAT := 16#0000, P := 9, OUT => "REVAMP".ALM13);
END_REGION

REGION Network 15
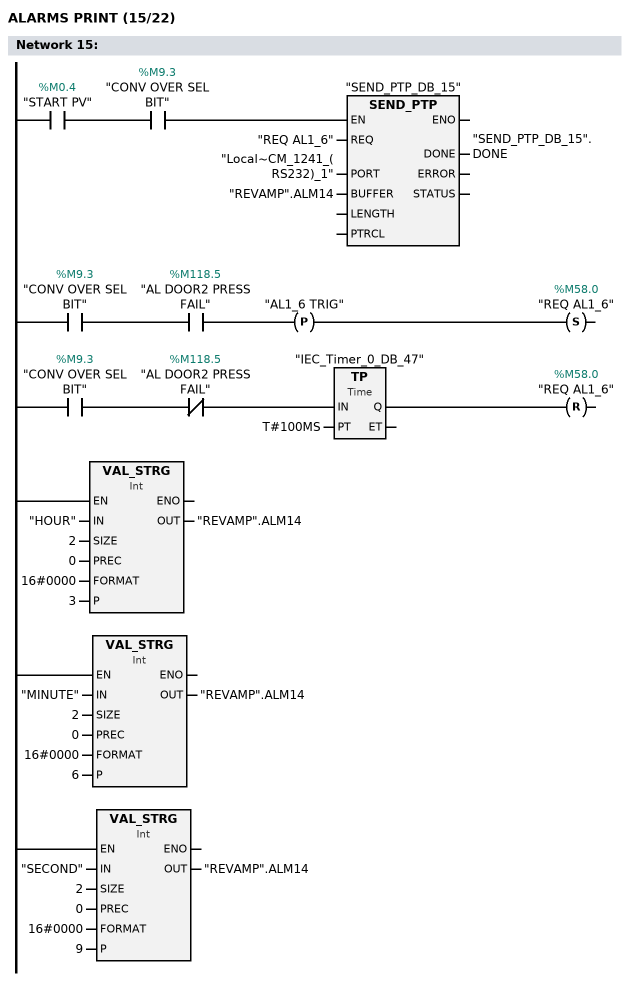
   RUNG wire#powerrail
      Contact( "START PV" )
      Contact( "CONV OVER SEL BIT" )
      "SEND_PTP_DB_15".SEND_PTP(REQ := "REQ AL1_6", PORT := "Local~CM_1241_(RS232)_1", BUFFER := "REVAMP".ALM14, LENGTH :=, PTRCL :=, DONE => "SEND_PTP_DB_15".DONE, ERROR =>, STATUS =>)
   END_RUNG
   RUNG wire#powerrail
      Contact( "CONV OVER SEL BIT" )
      Contact( "AL DOOR2 PRESS FAIL" )
      P_Trig( "AL1_6 TRIG" )
      S_Coil( "REQ AL1_6" )
   END_RUNG
   RUNG wire#powerrail
      Contact( "CONV OVER SEL BIT" )
      I_Contact( "AL DOOR2 PRESS FAIL" )
      { S7_Templates := "time_type := Time" } "IEC_Timer_0_DB_47".TP(pt := T#100MS, et =>)
      R_Coil( "REQ AL1_6" )
   END_RUNG
   RUNG wire#powerrail
      { S7_Templates := "[value_type := Int, str_type := String]" } VAL_STRG(IN := "HOUR", SIZE := 2, PREC := 0, FORMAT := 16#0000, P := 3, OUT => "REVAMP".ALM14)
   END_RUNG
   RUNG wire#powerrail
      { S7_Templates := "[value_type := Int, str_type := String]" } VAL_STRG(IN := "MINUTE", SIZE := 2, PREC := 0, FORMAT := 16#0000, P := 6, OUT => "REVAMP".ALM14)
   END_RUNG
   RUNG wire#powerrail
      { S7_Templates := "[value_type := Int, str_type := String]" } VAL_STRG(IN := "SECOND", SIZE := 2, PREC := 0, FORMAT := 16#0000, P := 9, OUT => "REVAMP".ALM14)
   END_RUNG
   // the same network as SCL:
   IF "START PV" AND "CONV OVER SEL BIT" THEN
       "SEND_PTP_DB_15"(REQ := "REQ AL1_6",   // SEND_PTP
                        PORT := "Local~CM_1241_(RS232)_1",
                        BUFFER := "REVAMP".ALM14,
                        DONE => "SEND_PTP_DB_15".DONE);
   END_IF;
   #_w1 := "CONV OVER SEL BIT" AND "AL DOOR2 PRESS FAIL";
   #_w2 := #_w1 AND NOT "AL1_6 TRIG";   // rising edge
   "AL1_6 TRIG" := #_w1;
   IF #_w2 THEN "REQ AL1_6" := TRUE; END_IF;
   "IEC_Timer_0_DB_47".TP(IN := "CONV OVER SEL BIT" AND NOT "AL DOOR2 PRESS FAIL", PT := T#100MS);
   IF "IEC_Timer_0_DB_47".Q THEN "REQ AL1_6" := FALSE; END_IF;
   VAL_STRG(IN := "HOUR", SIZE := 2, PREC := 0, FORMAT := 16#0000, P := 3, OUT => "REVAMP".ALM14);
   VAL_STRG(IN := "MINUTE", SIZE := 2, PREC := 0, FORMAT := 16#0000, P := 6, OUT => "REVAMP".ALM14);
   VAL_STRG(IN := "SECOND", SIZE := 2, PREC := 0, FORMAT := 16#0000, P := 9, OUT => "REVAMP".ALM14);
END_REGION

REGION Network 16
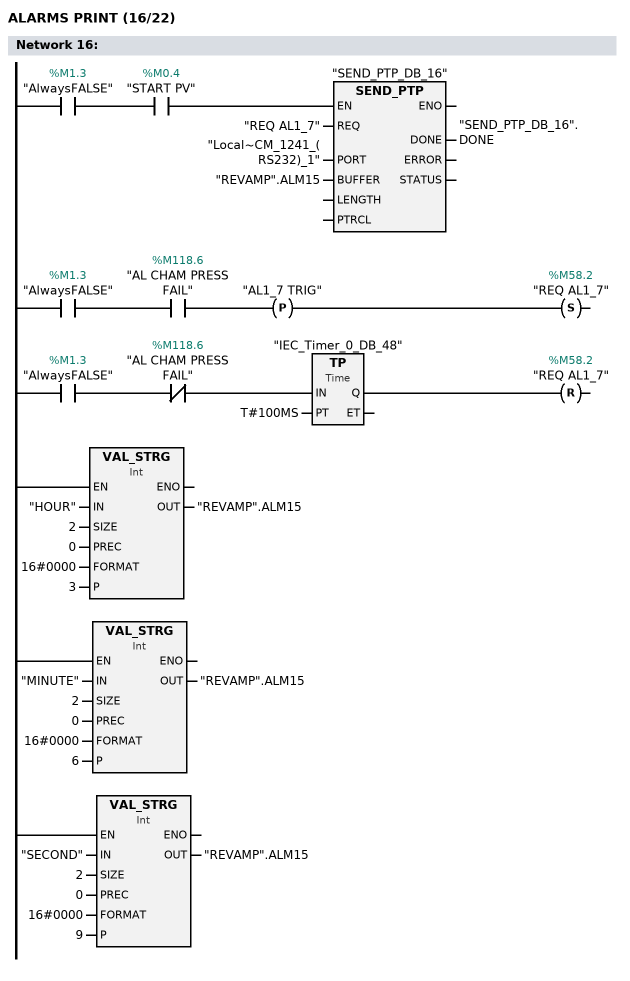
   RUNG wire#powerrail
      Contact( "AlwaysFALSE" )
      Contact( "START PV" )
      "SEND_PTP_DB_16".SEND_PTP(REQ := "REQ AL1_7", PORT := "Local~CM_1241_(RS232)_1", BUFFER := "REVAMP".ALM15, LENGTH :=, PTRCL :=, DONE => "SEND_PTP_DB_16".DONE, ERROR =>, STATUS =>)
   END_RUNG
   RUNG wire#powerrail
      Contact( "AlwaysFALSE" )
      Contact( "AL CHAM PRESS FAIL" )
      P_Trig( "AL1_7 TRIG" )
      S_Coil( "REQ AL1_7" )
   END_RUNG
   RUNG wire#powerrail
      Contact( "AlwaysFALSE" )
      I_Contact( "AL CHAM PRESS FAIL" )
      { S7_Templates := "time_type := Time" } "IEC_Timer_0_DB_48".TP(pt := T#100MS, et =>)
      R_Coil( "REQ AL1_7" )
   END_RUNG
   RUNG wire#powerrail
      { S7_Templates := "[value_type := Int, str_type := String]" } VAL_STRG(IN := "HOUR", SIZE := 2, PREC := 0, FORMAT := 16#0000, P := 3, OUT => "REVAMP".ALM15)
   END_RUNG
   RUNG wire#powerrail
      { S7_Templates := "[value_type := Int, str_type := String]" } VAL_STRG(IN := "MINUTE", SIZE := 2, PREC := 0, FORMAT := 16#0000, P := 6, OUT => "REVAMP".ALM15)
   END_RUNG
   RUNG wire#powerrail
      { S7_Templates := "[value_type := Int, str_type := String]" } VAL_STRG(IN := "SECOND", SIZE := 2, PREC := 0, FORMAT := 16#0000, P := 9, OUT => "REVAMP".ALM15)
   END_RUNG
   // the same network as SCL:
   IF "AlwaysFALSE" AND "START PV" THEN
       "SEND_PTP_DB_16"(REQ := "REQ AL1_7",   // SEND_PTP
                        PORT := "Local~CM_1241_(RS232)_1",
                        BUFFER := "REVAMP".ALM15,
                        DONE => "SEND_PTP_DB_16".DONE);
   END_IF;
   #_w1 := "AlwaysFALSE" AND "AL CHAM PRESS FAIL";
   #_w2 := #_w1 AND NOT "AL1_7 TRIG";   // rising edge
   "AL1_7 TRIG" := #_w1;
   IF #_w2 THEN "REQ AL1_7" := TRUE; END_IF;
   "IEC_Timer_0_DB_48".TP(IN := "AlwaysFALSE" AND NOT "AL CHAM PRESS FAIL", PT := T#100MS);
   IF "IEC_Timer_0_DB_48".Q THEN "REQ AL1_7" := FALSE; END_IF;
   VAL_STRG(IN := "HOUR", SIZE := 2, PREC := 0, FORMAT := 16#0000, P := 3, OUT => "REVAMP".ALM15);
   VAL_STRG(IN := "MINUTE", SIZE := 2, PREC := 0, FORMAT := 16#0000, P := 6, OUT => "REVAMP".ALM15);
   VAL_STRG(IN := "SECOND", SIZE := 2, PREC := 0, FORMAT := 16#0000, P := 9, OUT => "REVAMP".ALM15);
END_REGION

REGION Network 17
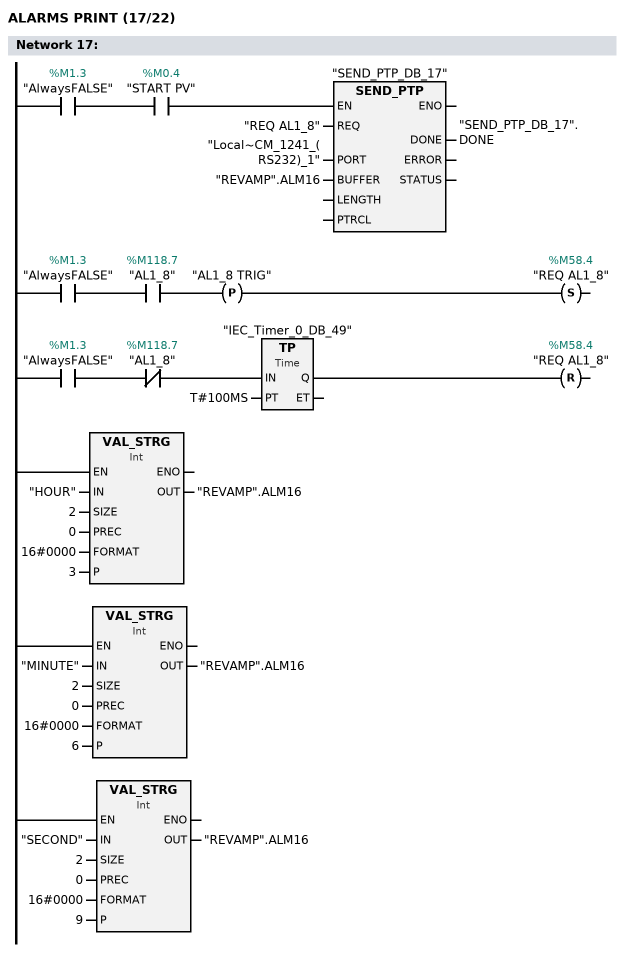
   RUNG wire#powerrail
      Contact( "AlwaysFALSE" )
      Contact( "START PV" )
      "SEND_PTP_DB_17".SEND_PTP(REQ := "REQ AL1_8", PORT := "Local~CM_1241_(RS232)_1", BUFFER := "REVAMP".ALM16, LENGTH :=, PTRCL :=, DONE => "SEND_PTP_DB_17".DONE, ERROR =>, STATUS =>)
   END_RUNG
   RUNG wire#powerrail
      Contact( "AlwaysFALSE" )
      Contact( "AL1_8" )
      P_Trig( "AL1_8 TRIG" )
      S_Coil( "REQ AL1_8" )
   END_RUNG
   RUNG wire#powerrail
      Contact( "AlwaysFALSE" )
      I_Contact( "AL1_8" )
      { S7_Templates := "time_type := Time" } "IEC_Timer_0_DB_49".TP(pt := T#100MS, et =>)
      R_Coil( "REQ AL1_8" )
   END_RUNG
   RUNG wire#powerrail
      { S7_Templates := "[value_type := Int, str_type := String]" } VAL_STRG(IN := "HOUR", SIZE := 2, PREC := 0, FORMAT := 16#0000, P := 3, OUT => "REVAMP".ALM16)
   END_RUNG
   RUNG wire#powerrail
      { S7_Templates := "[value_type := Int, str_type := String]" } VAL_STRG(IN := "MINUTE", SIZE := 2, PREC := 0, FORMAT := 16#0000, P := 6, OUT => "REVAMP".ALM16)
   END_RUNG
   RUNG wire#powerrail
      { S7_Templates := "[value_type := Int, str_type := String]" } VAL_STRG(IN := "SECOND", SIZE := 2, PREC := 0, FORMAT := 16#0000, P := 9, OUT => "REVAMP".ALM16)
   END_RUNG
   // the same network as SCL:
   IF "AlwaysFALSE" AND "START PV" THEN
       "SEND_PTP_DB_17"(REQ := "REQ AL1_8",   // SEND_PTP
                        PORT := "Local~CM_1241_(RS232)_1",
                        BUFFER := "REVAMP".ALM16,
                        DONE => "SEND_PTP_DB_17".DONE);
   END_IF;
   #_w1 := "AlwaysFALSE" AND "AL1_8";
   #_w2 := #_w1 AND NOT "AL1_8 TRIG";   // rising edge
   "AL1_8 TRIG" := #_w1;
   IF #_w2 THEN "REQ AL1_8" := TRUE; END_IF;
   "IEC_Timer_0_DB_49".TP(IN := "AlwaysFALSE" AND NOT "AL1_8", PT := T#100MS);
   IF "IEC_Timer_0_DB_49".Q THEN "REQ AL1_8" := FALSE; END_IF;
   VAL_STRG(IN := "HOUR", SIZE := 2, PREC := 0, FORMAT := 16#0000, P := 3, OUT => "REVAMP".ALM16);
   VAL_STRG(IN := "MINUTE", SIZE := 2, PREC := 0, FORMAT := 16#0000, P := 6, OUT => "REVAMP".ALM16);
   VAL_STRG(IN := "SECOND", SIZE := 2, PREC := 0, FORMAT := 16#0000, P := 9, OUT => "REVAMP".ALM16);
END_REGION

REGION Network 18
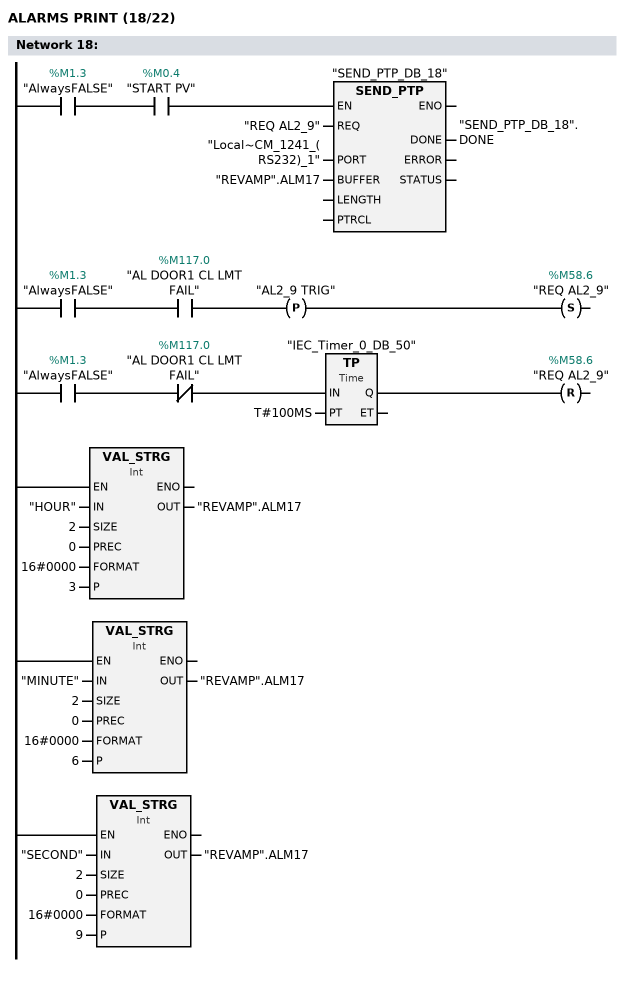
   RUNG wire#powerrail
      Contact( "AlwaysFALSE" )
      Contact( "START PV" )
      "SEND_PTP_DB_18".SEND_PTP(REQ := "REQ AL2_9", PORT := "Local~CM_1241_(RS232)_1", BUFFER := "REVAMP".ALM17, LENGTH :=, PTRCL :=, DONE => "SEND_PTP_DB_18".DONE, ERROR =>, STATUS =>)
   END_RUNG
   RUNG wire#powerrail
      Contact( "AlwaysFALSE" )
      Contact( "AL DOOR1 CL LMT FAIL" )
      P_Trig( "AL2_9 TRIG" )
      S_Coil( "REQ AL2_9" )
   END_RUNG
   RUNG wire#powerrail
      Contact( "AlwaysFALSE" )
      I_Contact( "AL DOOR1 CL LMT FAIL" )
      { S7_Templates := "time_type := Time" } "IEC_Timer_0_DB_50".TP(pt := T#100MS, et =>)
      R_Coil( "REQ AL2_9" )
   END_RUNG
   RUNG wire#powerrail
      { S7_Templates := "[value_type := Int, str_type := String]" } VAL_STRG(IN := "HOUR", SIZE := 2, PREC := 0, FORMAT := 16#0000, P := 3, OUT => "REVAMP".ALM17)
   END_RUNG
   RUNG wire#powerrail
      { S7_Templates := "[value_type := Int, str_type := String]" } VAL_STRG(IN := "MINUTE", SIZE := 2, PREC := 0, FORMAT := 16#0000, P := 6, OUT => "REVAMP".ALM17)
   END_RUNG
   RUNG wire#powerrail
      { S7_Templates := "[value_type := Int, str_type := String]" } VAL_STRG(IN := "SECOND", SIZE := 2, PREC := 0, FORMAT := 16#0000, P := 9, OUT => "REVAMP".ALM17)
   END_RUNG
   // the same network as SCL:
   IF "AlwaysFALSE" AND "START PV" THEN
       "SEND_PTP_DB_18"(REQ := "REQ AL2_9",   // SEND_PTP
                        PORT := "Local~CM_1241_(RS232)_1",
                        BUFFER := "REVAMP".ALM17,
                        DONE => "SEND_PTP_DB_18".DONE);
   END_IF;
   #_w1 := "AlwaysFALSE" AND "AL DOOR1 CL LMT FAIL";
   #_w2 := #_w1 AND NOT "AL2_9 TRIG";   // rising edge
   "AL2_9 TRIG" := #_w1;
   IF #_w2 THEN "REQ AL2_9" := TRUE; END_IF;
   "IEC_Timer_0_DB_50".TP(IN := "AlwaysFALSE" AND NOT "AL DOOR1 CL LMT FAIL", PT := T#100MS);
   IF "IEC_Timer_0_DB_50".Q THEN "REQ AL2_9" := FALSE; END_IF;
   VAL_STRG(IN := "HOUR", SIZE := 2, PREC := 0, FORMAT := 16#0000, P := 3, OUT => "REVAMP".ALM17);
   VAL_STRG(IN := "MINUTE", SIZE := 2, PREC := 0, FORMAT := 16#0000, P := 6, OUT => "REVAMP".ALM17);
   VAL_STRG(IN := "SECOND", SIZE := 2, PREC := 0, FORMAT := 16#0000, P := 9, OUT => "REVAMP".ALM17);
END_REGION

REGION Network 19
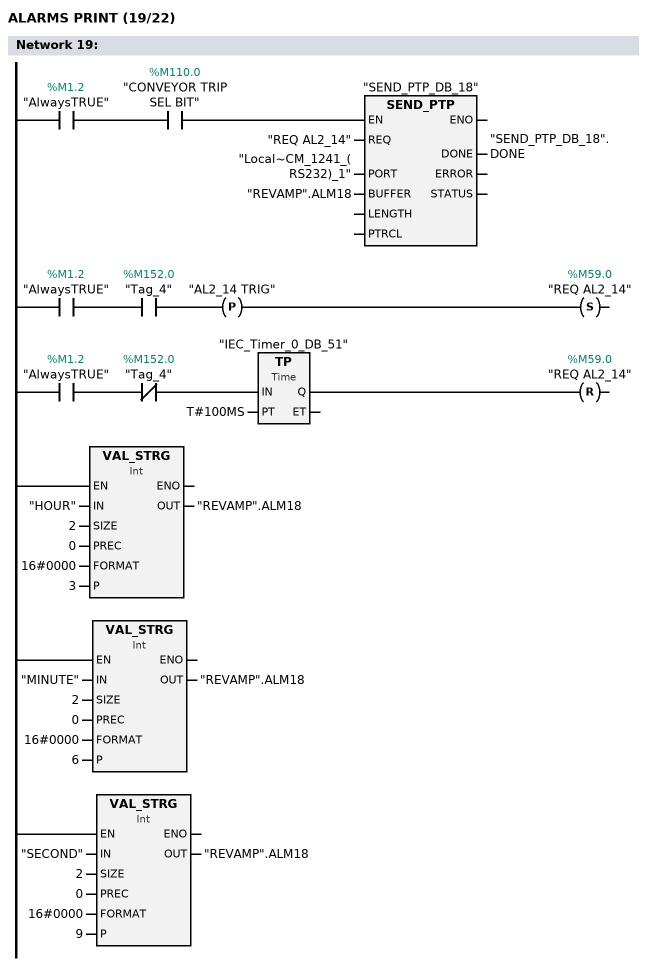
   RUNG wire#powerrail
      Contact( "AlwaysTRUE" )
      Contact( "CONVEYOR TRIP SEL BIT" )
      "SEND_PTP_DB_18".SEND_PTP(REQ := "REQ AL2_14", PORT := "Local~CM_1241_(RS232)_1", BUFFER := "REVAMP".ALM18, LENGTH :=, PTRCL :=, DONE => "SEND_PTP_DB_18".DONE, ERROR =>, STATUS =>)
   END_RUNG
   RUNG wire#powerrail
      Contact( "AlwaysTRUE" )
      Contact( "Tag_4" )
      P_Trig( "AL2_14 TRIG" )
      S_Coil( "REQ AL2_14" )
   END_RUNG
   RUNG wire#powerrail
      Contact( "AlwaysTRUE" )
      I_Contact( "Tag_4" )
      { S7_Templates := "time_type := Time" } "IEC_Timer_0_DB_51".TP(pt := T#100MS, et =>)
      R_Coil( "REQ AL2_14" )
   END_RUNG
   RUNG wire#powerrail
      { S7_Templates := "[value_type := Int, str_type := String]" } VAL_STRG(IN := "HOUR", SIZE := 2, PREC := 0, FORMAT := 16#0000, P := 3, OUT => "REVAMP".ALM18)
   END_RUNG
   RUNG wire#powerrail
      { S7_Templates := "[value_type := Int, str_type := String]" } VAL_STRG(IN := "MINUTE", SIZE := 2, PREC := 0, FORMAT := 16#0000, P := 6, OUT => "REVAMP".ALM18)
   END_RUNG
   RUNG wire#powerrail
      { S7_Templates := "[value_type := Int, str_type := String]" } VAL_STRG(IN := "SECOND", SIZE := 2, PREC := 0, FORMAT := 16#0000, P := 9, OUT => "REVAMP".ALM18)
   END_RUNG
   // the same network as SCL:
   IF "AlwaysTRUE" AND "CONVEYOR TRIP SEL BIT" THEN
       "SEND_PTP_DB_18"(REQ := "REQ AL2_14",   // SEND_PTP
                        PORT := "Local~CM_1241_(RS232)_1",
                        BUFFER := "REVAMP".ALM18,
                        DONE => "SEND_PTP_DB_18".DONE);
   END_IF;
   #_w1 := "AlwaysTRUE" AND "Tag_4";
   #_w2 := #_w1 AND NOT "AL2_14 TRIG";   // rising edge
   "AL2_14 TRIG" := #_w1;
   IF #_w2 THEN "REQ AL2_14" := TRUE; END_IF;
   "IEC_Timer_0_DB_51".TP(IN := "AlwaysTRUE" AND NOT "Tag_4", PT := T#100MS);
   IF "IEC_Timer_0_DB_51".Q THEN "REQ AL2_14" := FALSE; END_IF;
   VAL_STRG(IN := "HOUR", SIZE := 2, PREC := 0, FORMAT := 16#0000, P := 3, OUT => "REVAMP".ALM18);
   VAL_STRG(IN := "MINUTE", SIZE := 2, PREC := 0, FORMAT := 16#0000, P := 6, OUT => "REVAMP".ALM18);
   VAL_STRG(IN := "SECOND", SIZE := 2, PREC := 0, FORMAT := 16#0000, P := 9, OUT => "REVAMP".ALM18);
END_REGION

REGION Network 20
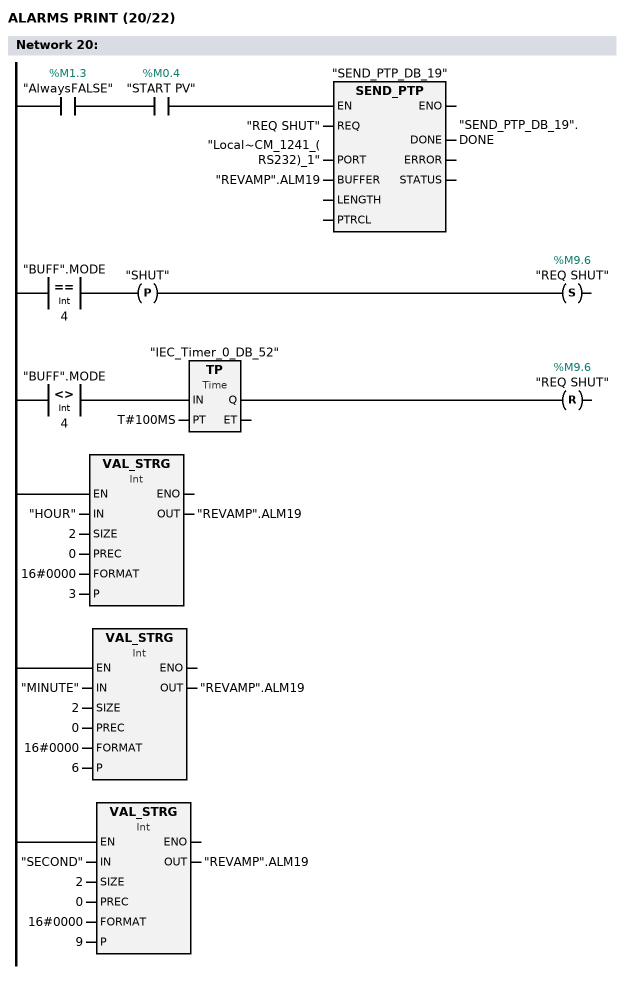
   RUNG wire#powerrail
      Contact( "AlwaysFALSE" )
      Contact( "START PV" )
      "SEND_PTP_DB_19".SEND_PTP(REQ := "REQ SHUT", PORT := "Local~CM_1241_(RS232)_1", BUFFER := "REVAMP".ALM19, LENGTH :=, PTRCL :=, DONE => "SEND_PTP_DB_19".DONE, ERROR =>, STATUS =>)
   END_RUNG
   RUNG wire#powerrail
      { S7_Templates := "SrcType := Int" } EQ_Contact(in1 := "BUFF".MODE, in2 := 4)
      P_Trig( "SHUT" )
      S_Coil( "REQ SHUT" )
   END_RUNG
   RUNG wire#powerrail
      { S7_Templates := "SrcType := Int" } NE_Contact(in1 := "BUFF".MODE, in2 := 4)
      { S7_Templates := "time_type := Time" } "IEC_Timer_0_DB_52".TP(pt := T#100MS, et =>)
      R_Coil( "REQ SHUT" )
   END_RUNG
   RUNG wire#powerrail
      { S7_Templates := "[value_type := Int, str_type := String]" } VAL_STRG(IN := "HOUR", SIZE := 2, PREC := 0, FORMAT := 16#0000, P := 3, OUT => "REVAMP".ALM19)
   END_RUNG
   RUNG wire#powerrail
      { S7_Templates := "[value_type := Int, str_type := String]" } VAL_STRG(IN := "MINUTE", SIZE := 2, PREC := 0, FORMAT := 16#0000, P := 6, OUT => "REVAMP".ALM19)
   END_RUNG
   RUNG wire#powerrail
      { S7_Templates := "[value_type := Int, str_type := String]" } VAL_STRG(IN := "SECOND", SIZE := 2, PREC := 0, FORMAT := 16#0000, P := 9, OUT => "REVAMP".ALM19)
   END_RUNG
   // the same network as SCL:
   IF "AlwaysFALSE" AND "START PV" THEN
       "SEND_PTP_DB_19"(REQ := "REQ SHUT",   // SEND_PTP
                        PORT := "Local~CM_1241_(RS232)_1",
                        BUFFER := "REVAMP".ALM19,
                        DONE => "SEND_PTP_DB_19".DONE);
   END_IF;
   #_w1 := "BUFF".MODE = 4;
   #_w2 := #_w1 AND NOT "SHUT";   // rising edge
   "SHUT" := #_w1;
   IF #_w2 THEN "REQ SHUT" := TRUE; END_IF;
   "IEC_Timer_0_DB_52".TP(IN := "BUFF".MODE <> 4, PT := T#100MS);
   IF "IEC_Timer_0_DB_52".Q THEN "REQ SHUT" := FALSE; END_IF;
   VAL_STRG(IN := "HOUR", SIZE := 2, PREC := 0, FORMAT := 16#0000, P := 3, OUT => "REVAMP".ALM19);
   VAL_STRG(IN := "MINUTE", SIZE := 2, PREC := 0, FORMAT := 16#0000, P := 6, OUT => "REVAMP".ALM19);
   VAL_STRG(IN := "SECOND", SIZE := 2, PREC := 0, FORMAT := 16#0000, P := 9, OUT => "REVAMP".ALM19);
END_REGION

REGION Network 21
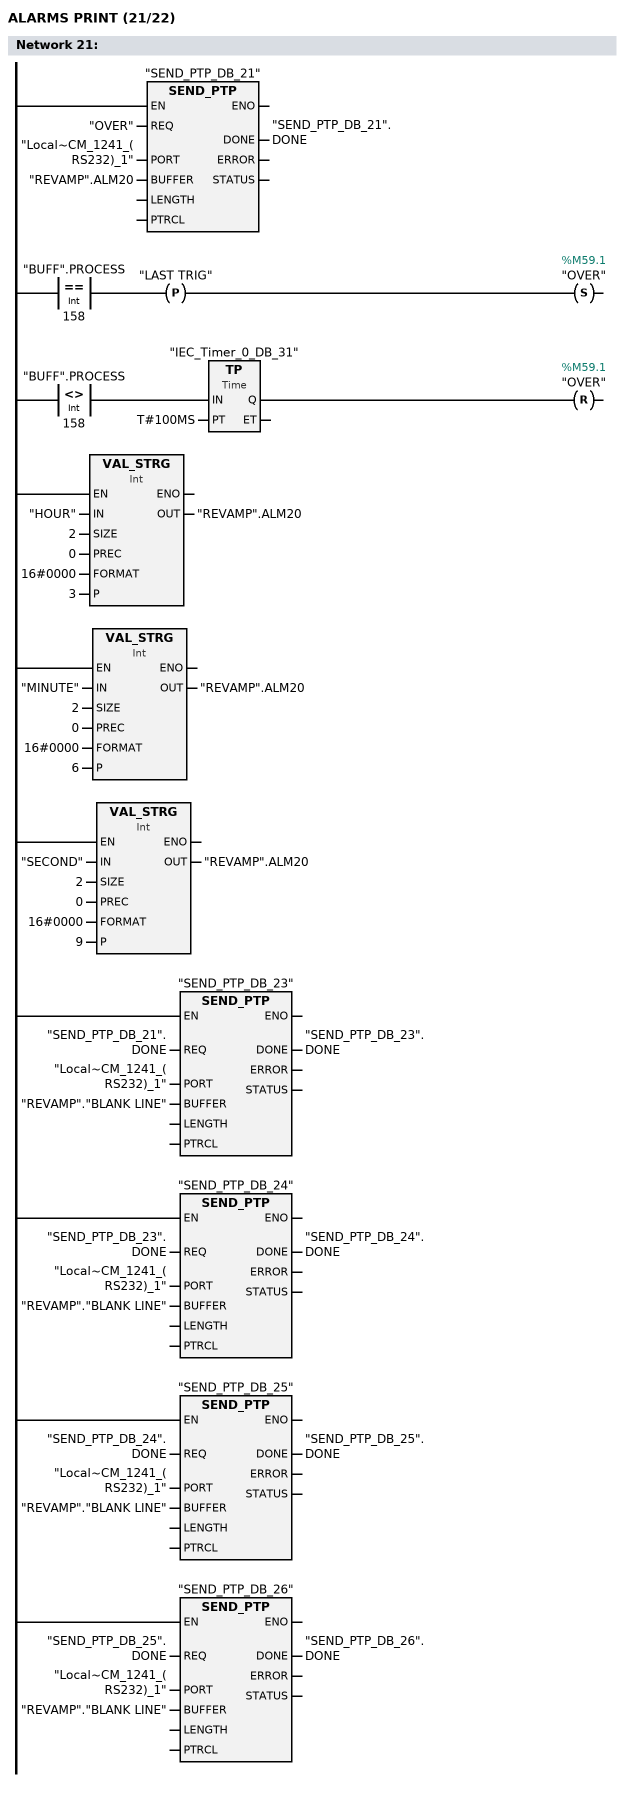
   RUNG wire#powerrail
      "SEND_PTP_DB_21".SEND_PTP(REQ := "OVER", PORT := "Local~CM_1241_(RS232)_1", BUFFER := "REVAMP".ALM20, LENGTH :=, PTRCL :=, DONE => "SEND_PTP_DB_21".DONE, ERROR =>, STATUS =>)
   END_RUNG
   RUNG wire#powerrail
      { S7_Templates := "SrcType := Int" } EQ_Contact(in1 := "BUFF".PROCESS, in2 := 158)
      P_Trig( "LAST TRIG" )
      S_Coil( "OVER" )
   END_RUNG
   RUNG wire#powerrail
      { S7_Templates := "SrcType := Int" } NE_Contact(in1 := "BUFF".PROCESS, in2 := 158)
      { S7_Templates := "time_type := Time" } "IEC_Timer_0_DB_31".TP(pt := T#100MS, et =>)
      R_Coil( "OVER" )
   END_RUNG
   RUNG wire#powerrail
      { S7_Templates := "[value_type := Int, str_type := String]" } VAL_STRG(IN := "HOUR", SIZE := 2, PREC := 0, FORMAT := 16#0000, P := 3, OUT => "REVAMP".ALM20)
   END_RUNG
   RUNG wire#powerrail
      { S7_Templates := "[value_type := Int, str_type := String]" } VAL_STRG(IN := "MINUTE", SIZE := 2, PREC := 0, FORMAT := 16#0000, P := 6, OUT => "REVAMP".ALM20)
   END_RUNG
   RUNG wire#powerrail
      { S7_Templates := "[value_type := Int, str_type := String]" } VAL_STRG(IN := "SECOND", SIZE := 2, PREC := 0, FORMAT := 16#0000, P := 9, OUT => "REVAMP".ALM20)
   END_RUNG
   RUNG wire#powerrail
      "SEND_PTP_DB_23".SEND_PTP(REQ := "SEND_PTP_DB_21".DONE, PORT := "Local~CM_1241_(RS232)_1", BUFFER := "REVAMP"."BLANK LINE", LENGTH :=, PTRCL :=, DONE => "SEND_PTP_DB_23".DONE, ERROR =>, STATUS =>)
   END_RUNG
   RUNG wire#powerrail
      "SEND_PTP_DB_24".SEND_PTP(REQ := "SEND_PTP_DB_23".DONE, PORT := "Local~CM_1241_(RS232)_1", BUFFER := "REVAMP"."BLANK LINE", LENGTH :=, PTRCL :=, DONE => "SEND_PTP_DB_24".DONE, ERROR =>, STATUS =>)
   END_RUNG
   RUNG wire#powerrail
      "SEND_PTP_DB_25".SEND_PTP(REQ := "SEND_PTP_DB_24".DONE, PORT := "Local~CM_1241_(RS232)_1", BUFFER := "REVAMP"."BLANK LINE", LENGTH :=, PTRCL :=, DONE => "SEND_PTP_DB_25".DONE, ERROR =>, STATUS =>)
   END_RUNG
   RUNG wire#powerrail
      "SEND_PTP_DB_26".SEND_PTP(REQ := "SEND_PTP_DB_25".DONE, PORT := "Local~CM_1241_(RS232)_1", BUFFER := "REVAMP"."BLANK LINE", LENGTH :=, PTRCL :=, DONE => "SEND_PTP_DB_26".DONE, ERROR =>, STATUS =>)
   END_RUNG
   // the same network as SCL:
   "SEND_PTP_DB_21"(REQ := "OVER",   // SEND_PTP
                    PORT := "Local~CM_1241_(RS232)_1",
                    BUFFER := "REVAMP".ALM20,
                    DONE => "SEND_PTP_DB_21".DONE);
   #_w1 := "BUFF".PROCESS = 158;
   #_w2 := #_w1 AND NOT "LAST TRIG";   // rising edge
   "LAST TRIG" := #_w1;
   IF #_w2 THEN "OVER" := TRUE; END_IF;
   "IEC_Timer_0_DB_31".TP(IN := "BUFF".PROCESS <> 158, PT := T#100MS);
   IF "IEC_Timer_0_DB_31".Q THEN "OVER" := FALSE; END_IF;
   VAL_STRG(IN := "HOUR", SIZE := 2, PREC := 0, FORMAT := 16#0000, P := 3, OUT => "REVAMP".ALM20);
   VAL_STRG(IN := "MINUTE", SIZE := 2, PREC := 0, FORMAT := 16#0000, P := 6, OUT => "REVAMP".ALM20);
   VAL_STRG(IN := "SECOND", SIZE := 2, PREC := 0, FORMAT := 16#0000, P := 9, OUT => "REVAMP".ALM20);
   "SEND_PTP_DB_23"(REQ := "SEND_PTP_DB_21".DONE,   // SEND_PTP
                    PORT := "Local~CM_1241_(RS232)_1",
                    BUFFER := "REVAMP"."BLANK LINE",
                    DONE => "SEND_PTP_DB_23".DONE);
   "SEND_PTP_DB_24"(REQ := "SEND_PTP_DB_23".DONE,   // SEND_PTP
                    PORT := "Local~CM_1241_(RS232)_1",
                    BUFFER := "REVAMP"."BLANK LINE",
                    DONE => "SEND_PTP_DB_24".DONE);
   "SEND_PTP_DB_25"(REQ := "SEND_PTP_DB_24".DONE,   // SEND_PTP
                    PORT := "Local~CM_1241_(RS232)_1",
                    BUFFER := "REVAMP"."BLANK LINE",
                    DONE => "SEND_PTP_DB_25".DONE);
   "SEND_PTP_DB_26"(REQ := "SEND_PTP_DB_25".DONE,   // SEND_PTP
                    PORT := "Local~CM_1241_(RS232)_1",
                    BUFFER := "REVAMP"."BLANK LINE",
                    DONE => "SEND_PTP_DB_26".DONE);
END_REGION

REGION Network 22
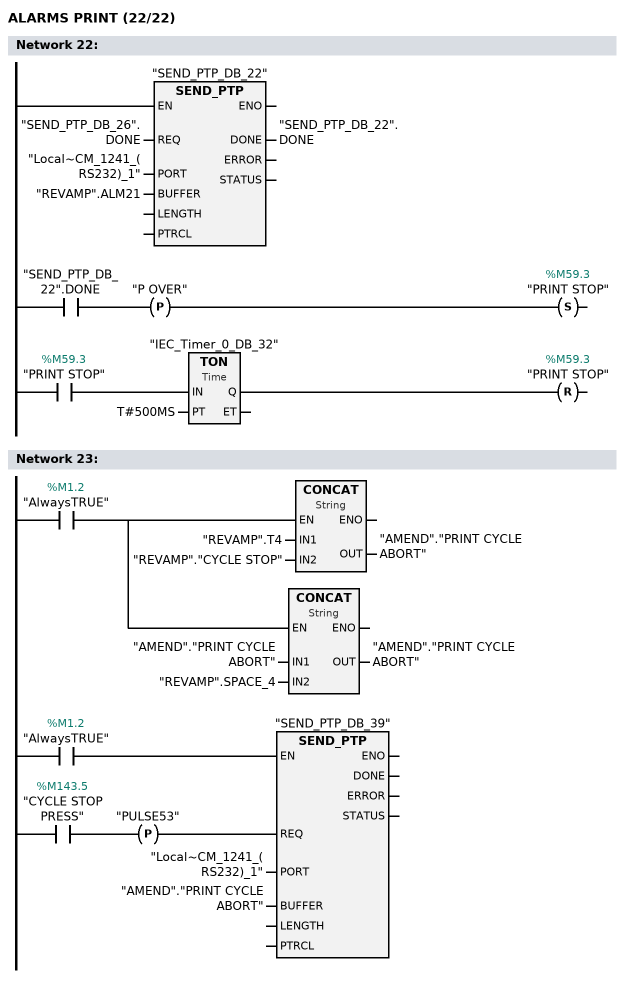
   RUNG wire#powerrail
      "SEND_PTP_DB_22".SEND_PTP(REQ := "SEND_PTP_DB_26".DONE, PORT := "Local~CM_1241_(RS232)_1", BUFFER := "REVAMP".ALM21, LENGTH :=, PTRCL :=, DONE => "SEND_PTP_DB_22".DONE, ERROR =>, STATUS =>)
   END_RUNG
   RUNG wire#powerrail
      Contact( "SEND_PTP_DB_22".DONE )
      P_Trig( "P OVER" )
      S_Coil( "PRINT STOP" )
   END_RUNG
   RUNG wire#powerrail
      Contact( "PRINT STOP" )
      { S7_Templates := "time_type := Time" } "IEC_Timer_0_DB_32".TON(pt := T#500MS, et =>)
      R_Coil( "PRINT STOP" )
   END_RUNG
   // the same network as SCL:
   "SEND_PTP_DB_22"(REQ := "SEND_PTP_DB_26".DONE,   // SEND_PTP
                    PORT := "Local~CM_1241_(RS232)_1",
                    BUFFER := "REVAMP".ALM21,
                    DONE => "SEND_PTP_DB_22".DONE);
   #_w1 := "SEND_PTP_DB_22".DONE AND NOT "P OVER";   // rising edge
   "P OVER" := "SEND_PTP_DB_22".DONE;
   IF #_w1 THEN "PRINT STOP" := TRUE; END_IF;
   "IEC_Timer_0_DB_32".TON(IN := "PRINT STOP", PT := T#500MS);
   IF "IEC_Timer_0_DB_32".Q THEN "PRINT STOP" := FALSE; END_IF;
END_REGION

REGION Network 23
   RUNG wire#powerrail
      Contact( "AlwaysTRUE" )
      wire#w1
      { S7_Templates := "[card := 2, str_type := String]" } CONCAT(IN1 := "REVAMP".T4, IN2 := "REVAMP"."CYCLE STOP", OUT => "AMEND"."PRINT CYCLE ABORT")
   END_RUNG
   RUNG wire#w1
      { S7_Templates := "[card := 2, str_type := String]" } CONCAT(IN1 := "AMEND"."PRINT CYCLE ABORT", IN2 := "REVAMP".SPACE_4, OUT => "AMEND"."PRINT CYCLE ABORT")
   END_RUNG
   RUNG wire#powerrail
      Contact( "AlwaysTRUE" )
      "SEND_PTP_DB_39".SEND_PTP(REQ := wire#w2, PORT := "Local~CM_1241_(RS232)_1", BUFFER := "AMEND"."PRINT CYCLE ABORT", LENGTH :=, PTRCL :=, DONE =>, ERROR =>, STATUS =>)
   END_RUNG
   RUNG wire#powerrail
      Contact( "CYCLE STOP PRESS" )
      P_Trig( "PULSE53" )
   END_RUNG wire#w2
   // the same network as SCL:
   #_w1 := "AlwaysTRUE";
   IF #_w1 THEN
       CONCAT(IN1 := "REVAMP".T4, IN2 := "REVAMP"."CYCLE STOP", OUT => "AMEND"."PRINT CYCLE ABORT");
       CONCAT(IN1 := "AMEND"."PRINT CYCLE ABORT", IN2 := "REVAMP".SPACE_4, OUT => "AMEND"."PRINT CYCLE ABORT");
   END_IF;
   #_w2 := "CYCLE STOP PRESS" AND NOT "PULSE53";   // rising edge
   "PULSE53" := "CYCLE STOP PRESS";
   IF "AlwaysTRUE" THEN
       "SEND_PTP_DB_39"(REQ := #_w2, PORT := "Local~CM_1241_(RS232)_1", BUFFER := "AMEND"."PRINT CYCLE ABORT");   // SEND_PTP
   END_IF;
END_REGION
END_FUNCTION

FUNCTION "ALARMS" : Void   // FC8, LAD
{ S7_Optimized_Access := 'TRUE' }
// stored: SetENOAutomatically false
   VAR_TEMP   // added for the SCL form of the ladder/FBD networks
      _w1 : Bool;
      _w2 : Bool;
      _w3 : Bool;
      _w4 : Bool;
   END_VAR
BEGIN

REGION Network 1: ERROR
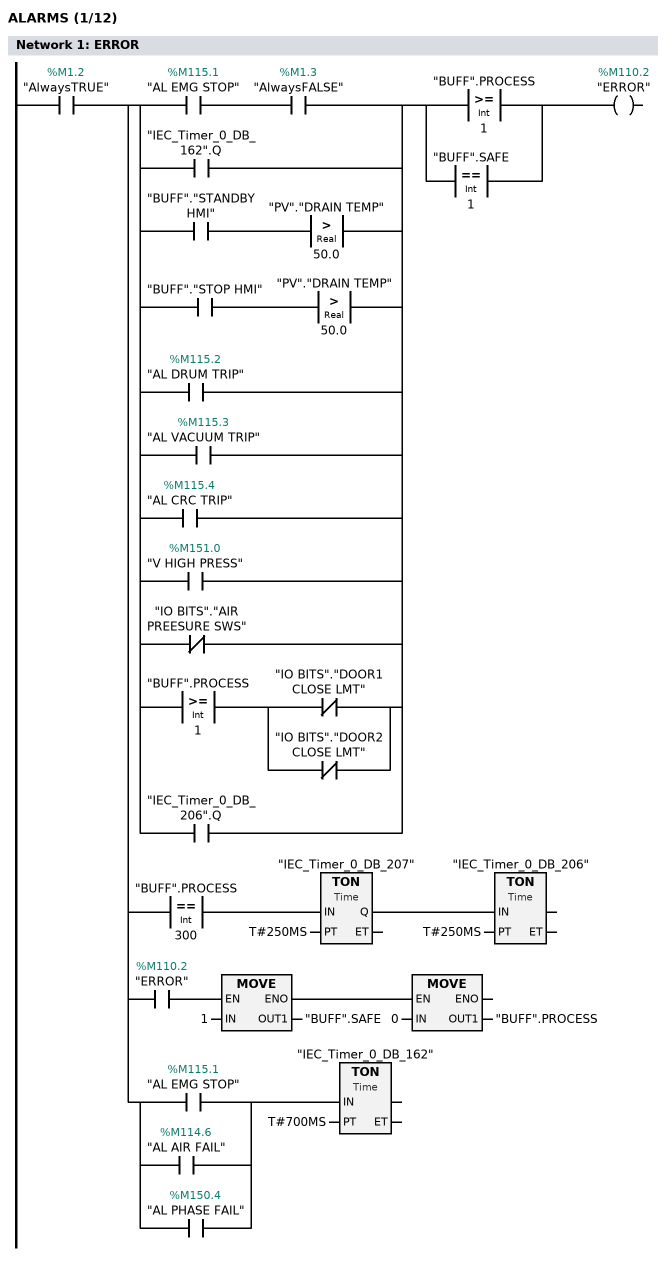
   RUNG wire#powerrail
      Contact( "AlwaysTRUE" )
      wire#w1
      Contact( "AL EMG STOP" )
      Contact( "AlwaysFALSE" )
      wire#w2
      { S7_Templates := "SrcType := Int" } GE_Contact(in1 := "BUFF".PROCESS, in2 := 1)
      wire#w4
      Coil( "ERROR" )
   END_RUNG
   RUNG wire#w1
      Contact( "IEC_Timer_0_DB_162".Q )
   END_RUNG wire#w2
   RUNG wire#w1
      Contact( "BUFF"."STANDBY HMI" )
      { S7_Templates := "SrcType := Real" } GT_Contact(in1 := "PV"."DRAIN TEMP", in2 := 50.0)
   END_RUNG wire#w2
   RUNG wire#w1
      Contact( "BUFF"."STOP HMI" )
      { S7_Templates := "SrcType := Real" } GT_Contact(in1 := "PV"."DRAIN TEMP", in2 := 50.0)
   END_RUNG wire#w2
   RUNG wire#w1
      Contact( "AL DRUM TRIP" )
   END_RUNG wire#w2
   RUNG wire#w1
      Contact( "AL VACUUM TRIP" )
   END_RUNG wire#w2
   RUNG wire#w1
      Contact( "AL CRC TRIP" )
   END_RUNG wire#w2
   RUNG wire#w1
      Contact( "V HIGH PRESS" )
   END_RUNG wire#w2
   RUNG wire#w1
      I_Contact( "IO BITS"."AIR PREESURE SWS" )
   END_RUNG wire#w2
   RUNG wire#w1
      { S7_Templates := "SrcType := Int" } GE_Contact(in1 := "BUFF".PROCESS, in2 := 1)
      wire#w3
      I_Contact( "IO BITS"."DOOR1 CLOSE LMT" )
   END_RUNG wire#w2
   RUNG wire#w3
      I_Contact( "IO BITS"."DOOR2 CLOSE LMT" )
   END_RUNG wire#w2
   RUNG wire#w1
      Contact( "IEC_Timer_0_DB_206".Q )
   END_RUNG wire#w2
   RUNG wire#w2
      { S7_Templates := "SrcType := Int" } EQ_Contact(in1 := "BUFF".SAFE, in2 := 1)
   END_RUNG wire#w4
   RUNG wire#w1
      { S7_Templates := "SrcType := Int" } EQ_Contact(in1 := "BUFF".PROCESS, in2 := 300)
      { S7_Templates := "time_type := Time" } "IEC_Timer_0_DB_207".TON(pt := T#250MS, et =>)
      { S7_Templates := "time_type := Time" } "IEC_Timer_0_DB_206".TON(pt := T#250MS, et =>)
   END_RUNG
   RUNG wire#w1
      Contact( "ERROR" )
      Move(in := 1, out1 => "BUFF".SAFE)
      Move(in := 0, out1 => "BUFF".PROCESS)
   END_RUNG
   RUNG wire#w1
      Contact( "AL EMG STOP" )
      wire#w5
      { S7_Templates := "time_type := Time" } "IEC_Timer_0_DB_162".TON(pt := T#700MS, et =>)
   END_RUNG
   RUNG wire#w1
      Contact( "AL AIR FAIL" )
   END_RUNG wire#w5
   RUNG wire#w1
      Contact( "AL PHASE FAIL" )
   END_RUNG wire#w5
   // the same network as SCL:
   "ERROR" := "AlwaysTRUE" AND (("AL EMG STOP" AND "AlwaysFALSE") OR "IEC_Timer_0_DB_162".Q OR ("BUFF"."STANDBY HMI" AND ("PV"."DRAIN TEMP" > 50.0)) OR ("BUFF"."STOP HMI" AND ("PV"."DRAIN TEMP" > 50.0)) OR "AL DRUM TRIP" OR "AL VACUUM TRIP" OR "AL CRC TRIP" OR "V HIGH PRESS" OR NOT "IO BITS"."AIR PREESURE SWS" OR (("BUFF".PROCESS >= 1) AND (NOT "IO BITS"."DOOR1 CLOSE LMT" OR NOT "IO BITS"."DOOR2 CLOSE LMT")) OR "IEC_Timer_0_DB_206".Q) AND (("BUFF".PROCESS >= 1) OR ("BUFF".SAFE = 1));
   "IEC_Timer_0_DB_207".TON(IN := "AlwaysTRUE" AND ("BUFF".PROCESS = 300), PT := T#250MS);
   "IEC_Timer_0_DB_206".TON(IN := "IEC_Timer_0_DB_207".Q, PT := T#250MS);
   IF "AlwaysTRUE" AND "ERROR" THEN
       "BUFF".SAFE := 1;
       "BUFF".PROCESS := 0;
   END_IF;
   "IEC_Timer_0_DB_162".TON(IN := "AlwaysTRUE" AND ("AL EMG STOP" OR "AL AIR FAIL" OR "AL PHASE FAIL"),
                           PT := T#700MS);
END_REGION

REGION Network 2: PFR
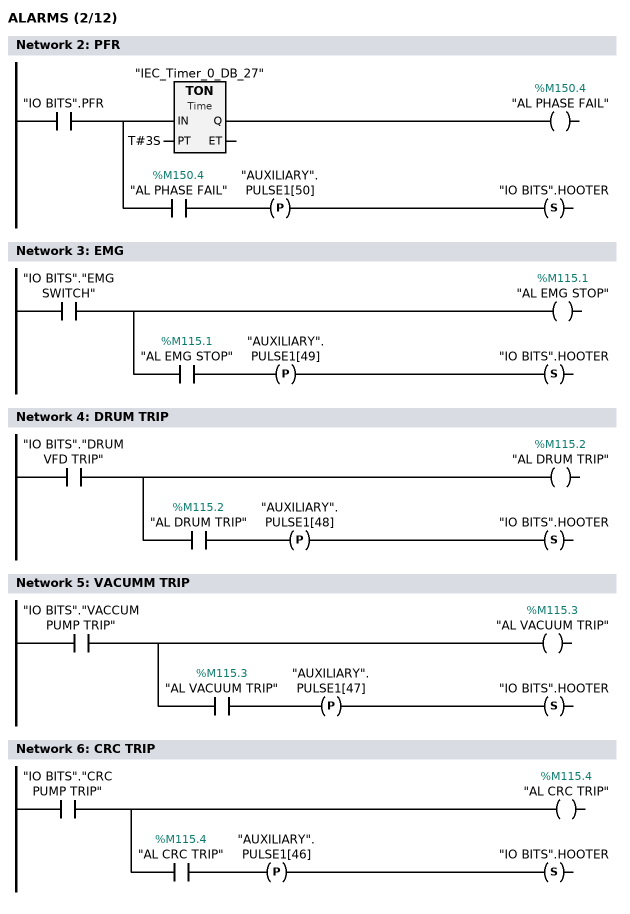
   RUNG wire#powerrail
      Contact( "IO BITS".PFR )
      wire#w1
      { S7_Templates := "time_type := Time" } "IEC_Timer_0_DB_27".TON(pt := T#3S, et =>)
      Coil( "AL PHASE FAIL" )
   END_RUNG
   RUNG wire#w1
      Contact( "AL PHASE FAIL" )
      P_Trig( "AUXILIARY".PULSE1[50] )
      S_Coil( "IO BITS".HOOTER )
   END_RUNG
   // the same network as SCL:
   "IEC_Timer_0_DB_27".TON(IN := "IO BITS".PFR, PT := T#3S);
   "AL PHASE FAIL" := "IEC_Timer_0_DB_27".Q;
   #_w1 := "IO BITS".PFR AND "AL PHASE FAIL";
   #_w2 := #_w1 AND NOT "AUXILIARY".PULSE1[50];   // rising edge
   "AUXILIARY".PULSE1[50] := #_w1;
   IF #_w2 THEN "IO BITS".HOOTER := TRUE; END_IF;
END_REGION

REGION Network 3: EMG
   RUNG wire#powerrail
      Contact( "IO BITS"."EMG SWITCH" )
      wire#w1
      Coil( "AL EMG STOP" )
   END_RUNG
   RUNG wire#w1
      Contact( "AL EMG STOP" )
      P_Trig( "AUXILIARY".PULSE1[49] )
      S_Coil( "IO BITS".HOOTER )
   END_RUNG
   // the same network as SCL:
   "AL EMG STOP" := "IO BITS"."EMG SWITCH";
   #_w1 := "IO BITS"."EMG SWITCH" AND "AL EMG STOP";
   #_w2 := #_w1 AND NOT "AUXILIARY".PULSE1[49];   // rising edge
   "AUXILIARY".PULSE1[49] := #_w1;
   IF #_w2 THEN "IO BITS".HOOTER := TRUE; END_IF;
END_REGION

REGION Network 4: DRUM TRIP
   RUNG wire#powerrail
      Contact( "IO BITS"."DRUM VFD TRIP" )
      wire#w1
      Coil( "AL DRUM TRIP" )
   END_RUNG
   RUNG wire#w1
      Contact( "AL DRUM TRIP" )
      P_Trig( "AUXILIARY".PULSE1[48] )
      S_Coil( "IO BITS".HOOTER )
   END_RUNG
   // the same network as SCL:
   "AL DRUM TRIP" := "IO BITS"."DRUM VFD TRIP";
   #_w1 := "IO BITS"."DRUM VFD TRIP" AND "AL DRUM TRIP";
   #_w2 := #_w1 AND NOT "AUXILIARY".PULSE1[48];   // rising edge
   "AUXILIARY".PULSE1[48] := #_w1;
   IF #_w2 THEN "IO BITS".HOOTER := TRUE; END_IF;
END_REGION

REGION Network 5: VACUMM TRIP
   RUNG wire#powerrail
      Contact( "IO BITS"."VACCUM PUMP TRIP" )
      wire#w1
      Coil( "AL VACUUM TRIP" )
   END_RUNG
   RUNG wire#w1
      Contact( "AL VACUUM TRIP" )
      P_Trig( "AUXILIARY".PULSE1[47] )
      S_Coil( "IO BITS".HOOTER )
   END_RUNG
   // the same network as SCL:
   "AL VACUUM TRIP" := "IO BITS"."VACCUM PUMP TRIP";
   #_w1 := "IO BITS"."VACCUM PUMP TRIP" AND "AL VACUUM TRIP";
   #_w2 := #_w1 AND NOT "AUXILIARY".PULSE1[47];   // rising edge
   "AUXILIARY".PULSE1[47] := #_w1;
   IF #_w2 THEN "IO BITS".HOOTER := TRUE; END_IF;
END_REGION

REGION Network 6: CRC TRIP
   RUNG wire#powerrail
      Contact( "IO BITS"."CRC PUMP TRIP" )
      wire#w1
      Coil( "AL CRC TRIP" )
   END_RUNG
   RUNG wire#w1
      Contact( "AL CRC TRIP" )
      P_Trig( "AUXILIARY".PULSE1[46] )
      S_Coil( "IO BITS".HOOTER )
   END_RUNG
   // the same network as SCL:
   "AL CRC TRIP" := "IO BITS"."CRC PUMP TRIP";
   #_w1 := "IO BITS"."CRC PUMP TRIP" AND "AL CRC TRIP";
   #_w2 := #_w1 AND NOT "AUXILIARY".PULSE1[46];   // rising edge
   "AUXILIARY".PULSE1[46] := #_w1;
   IF #_w2 THEN "IO BITS".HOOTER := TRUE; END_IF;
END_REGION

REGION Network 7: PROCESS START AND OVER
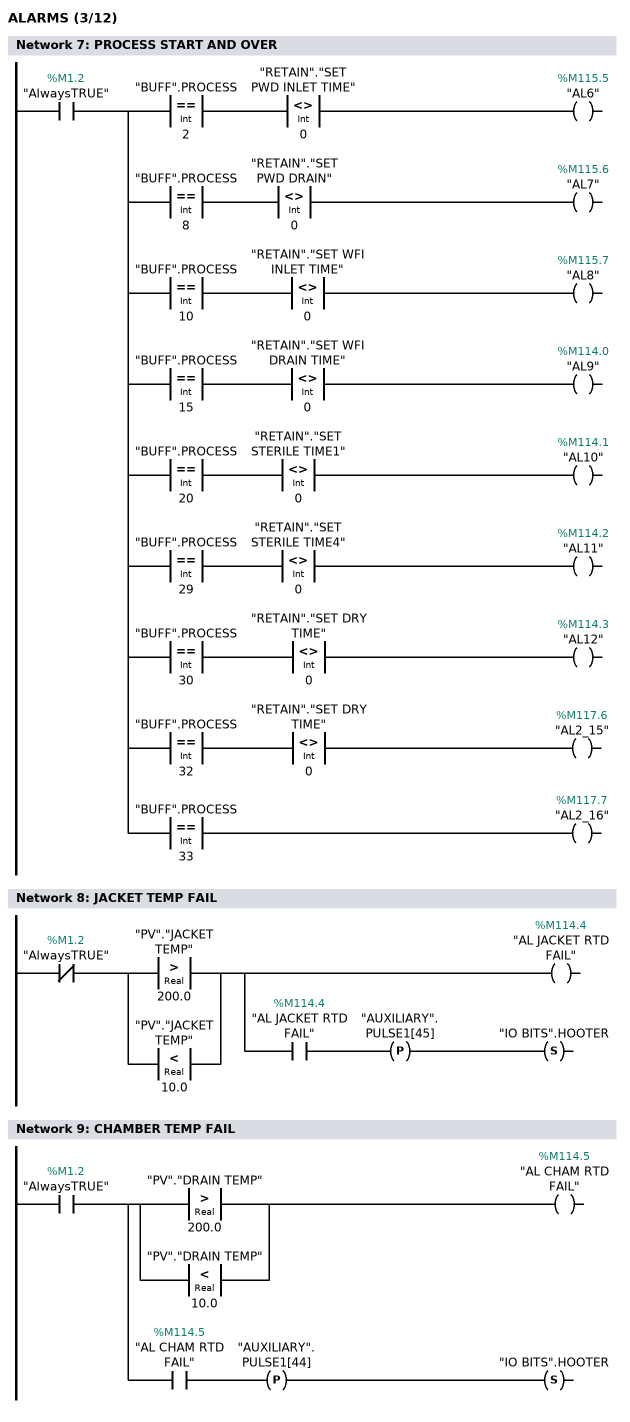
   RUNG wire#powerrail
      Contact( "AlwaysTRUE" )
      wire#w1
      { S7_Templates := "SrcType := Int" } EQ_Contact(in1 := "BUFF".PROCESS, in2 := 2)
      { S7_Templates := "SrcType := Int" } NE_Contact(in1 := "RETAIN"."SET PWD INLET TIME", in2 := 0)
      Coil( "AL6" )
   END_RUNG
   RUNG wire#w1
      { S7_Templates := "SrcType := Int" } EQ_Contact(in1 := "BUFF".PROCESS, in2 := 8)
      { S7_Templates := "SrcType := Int" } NE_Contact(in1 := "RETAIN"."SET PWD DRAIN", in2 := 0)
      Coil( "AL7" )
   END_RUNG
   RUNG wire#w1
      { S7_Templates := "SrcType := Int" } EQ_Contact(in1 := "BUFF".PROCESS, in2 := 10)
      { S7_Templates := "SrcType := Int" } NE_Contact(in1 := "RETAIN"."SET WFI INLET TIME", in2 := 0)
      Coil( "AL8" )
   END_RUNG
   RUNG wire#w1
      { S7_Templates := "SrcType := Int" } EQ_Contact(in1 := "BUFF".PROCESS, in2 := 15)
      { S7_Templates := "SrcType := Int" } NE_Contact(in1 := "RETAIN"."SET WFI DRAIN TIME", in2 := 0)
      Coil( "AL9" )
   END_RUNG
   RUNG wire#w1
      { S7_Templates := "SrcType := Int" } EQ_Contact(in1 := "BUFF".PROCESS, in2 := 20)
      { S7_Templates := "SrcType := Int" } NE_Contact(in1 := "RETAIN"."SET STERILE TIME1", in2 := 0)
      Coil( "AL10" )
   END_RUNG
   RUNG wire#w1
      { S7_Templates := "SrcType := Int" } EQ_Contact(in1 := "BUFF".PROCESS, in2 := 29)
      { S7_Templates := "SrcType := Int" } NE_Contact(in1 := "RETAIN"."SET STERILE TIME4", in2 := 0)
      Coil( "AL11" )
   END_RUNG
   RUNG wire#w1
      { S7_Templates := "SrcType := Int" } EQ_Contact(in1 := "BUFF".PROCESS, in2 := 30)
      { S7_Templates := "SrcType := Int" } NE_Contact(in1 := "RETAIN"."SET DRY TIME", in2 := 0)
      Coil( "AL12" )
   END_RUNG
   RUNG wire#w1
      { S7_Templates := "SrcType := Int" } EQ_Contact(in1 := "BUFF".PROCESS, in2 := 32)
      { S7_Templates := "SrcType := Int" } NE_Contact(in1 := "RETAIN"."SET DRY TIME", in2 := 0)
      Coil( "AL2_15" )
   END_RUNG
   RUNG wire#w1
      { S7_Templates := "SrcType := Int" } EQ_Contact(in1 := "BUFF".PROCESS, in2 := 33)
      Coil( "AL2_16" )
   END_RUNG
   // the same network as SCL:
   "AL6" := "AlwaysTRUE" AND ("BUFF".PROCESS = 2) AND ("RETAIN"."SET PWD INLET TIME" <> 0);
   "AL7" := "AlwaysTRUE" AND ("BUFF".PROCESS = 8) AND ("RETAIN"."SET PWD DRAIN" <> 0);
   "AL8" := "AlwaysTRUE" AND ("BUFF".PROCESS = 10) AND ("RETAIN"."SET WFI INLET TIME" <> 0);
   "AL9" := "AlwaysTRUE" AND ("BUFF".PROCESS = 15) AND ("RETAIN"."SET WFI DRAIN TIME" <> 0);
   "AL10" := "AlwaysTRUE" AND ("BUFF".PROCESS = 20) AND ("RETAIN"."SET STERILE TIME1" <> 0);
   "AL11" := "AlwaysTRUE" AND ("BUFF".PROCESS = 29) AND ("RETAIN"."SET STERILE TIME4" <> 0);
   "AL12" := "AlwaysTRUE" AND ("BUFF".PROCESS = 30) AND ("RETAIN"."SET DRY TIME" <> 0);
   "AL2_15" := "AlwaysTRUE" AND ("BUFF".PROCESS = 32) AND ("RETAIN"."SET DRY TIME" <> 0);
   "AL2_16" := "AlwaysTRUE" AND ("BUFF".PROCESS = 33);
END_REGION

REGION Network 8: JACKET TEMP FAIL
   RUNG wire#powerrail
      I_Contact( "AlwaysTRUE" )
      wire#w1
      { S7_Templates := "SrcType := Real" } GT_Contact(in1 := "PV"."JACKET TEMP", in2 := 200.0)
      wire#w2
      Coil( "AL JACKET RTD FAIL" )
   END_RUNG
   RUNG wire#w1
      { S7_Templates := "SrcType := Real" } LT_Contact(in1 := "PV"."JACKET TEMP", in2 := 10.0)
   END_RUNG wire#w2
   RUNG wire#w2
      Contact( "AL JACKET RTD FAIL" )
      P_Trig( "AUXILIARY".PULSE1[45] )
      S_Coil( "IO BITS".HOOTER )
   END_RUNG
   // the same network as SCL:
   "AL JACKET RTD FAIL" := NOT "AlwaysTRUE" AND (("PV"."JACKET TEMP" > 200.0) OR ("PV"."JACKET TEMP" < 10.0));
   #_w1 := "AL JACKET RTD FAIL" AND "AL JACKET RTD FAIL";
   #_w2 := #_w1 AND NOT "AUXILIARY".PULSE1[45];   // rising edge
   "AUXILIARY".PULSE1[45] := #_w1;
   IF #_w2 THEN "IO BITS".HOOTER := TRUE; END_IF;
END_REGION

REGION Network 9: CHAMBER TEMP FAIL
   RUNG wire#powerrail
      Contact( "AlwaysTRUE" )
      wire#w1
      { S7_Templates := "SrcType := Real" } GT_Contact(in1 := "PV"."DRAIN TEMP", in2 := 200.0)
      wire#w2
      Coil( "AL CHAM RTD FAIL" )
   END_RUNG
   RUNG wire#w1
      { S7_Templates := "SrcType := Real" } LT_Contact(in1 := "PV"."DRAIN TEMP", in2 := 10.0)
   END_RUNG wire#w2
   RUNG wire#w1
      Contact( "AL CHAM RTD FAIL" )
      P_Trig( "AUXILIARY".PULSE1[44] )
      S_Coil( "IO BITS".HOOTER )
   END_RUNG
   // the same network as SCL:
   "AL CHAM RTD FAIL" := "AlwaysTRUE" AND (("PV"."DRAIN TEMP" > 200.0) OR ("PV"."DRAIN TEMP" < 10.0));
   #_w1 := "AlwaysTRUE" AND "AL CHAM RTD FAIL";
   #_w2 := #_w1 AND NOT "AUXILIARY".PULSE1[44];   // rising edge
   "AUXILIARY".PULSE1[44] := #_w1;
   IF #_w2 THEN "IO BITS".HOOTER := TRUE; END_IF;
END_REGION

REGION Network 10: AIR FAIL
